FUNCTION_BLOCK TFCalcoliFuoriIngombriColonne
VAR_INPUT
	Traiettoria : POINTER TO TFTraiettoria;
	WorkSpace : POINTER TO TFMachinePalletizer_WorkSpace;
	WorkFootprint : POINTER TO ARRAY [1..MAXFOOTPRINT] OF TFMachinePalletizer_WorkFootprint; //Ingombri
	WorkPickPoint : POINTER TO ARRAY [1..MAXPICKPOINT] OF TFMachinePalletizer_WorkPickPoint;
	//WorkPickPointState : POINTER TO ARRAY [1..MAXPICKPOINT] OF TFMachinePalletizer_WorkPickPointState;
	WorkArea : POINTER TO ARRAY [1..MAXAREA] OF TFMachinePalletizer_WorkArea;
	WorkAreaState : POINTER TO ARRAY [1..MAXAREA] OF TFMachinePalletizer_WorkAreaState;
	Pallet : POINTER TO ARRAY [1..MAXPALLET] OF TFMachinePalletizer_Pallet;
	Layer : POINTER TO ARRAY [1..MAXLAYER] OF TFMachinePalletizer_Layer;
	Forming : POINTER TO ARRAY [1..MAXFORMING] OF TFMachinePalletizer_FormingForSlab;
	PickPlaceParameters	: POINTER TO TFMachinePalletizer_ParametersFromHMI;
	Mission : POINTER TO TFMachinePalletizer_Mission;
	
	WorkAreaManager : POINTER TO TFWorkAreaManager;
	ModuleAX_X : POINTER TO TFModulePalletizer_Ax;
	ModuleAX_Y : POINTER TO TFModulePalletizer_Ax;
	ModuleAX_Z : POINTER TO TFModulePalletizer_Ax;
	ModuleAX_J : POINTER TO TFModulePalletizer_Ax;
	ModuleAX_K : POINTER TO TFModulePalletizer_Ax;
	AbilitaCalcoloIngombroOttimizzato : BOOL := TRUE; //Abilitazione dell'utilizzo degli ingombri ottimizzati... calcoli in base all'angolo di rotazione della pinza
END_VAR
VAR
	f : INT;
	a : INT;
	P : INT;
	wa : int;
	waDXSX : INT;
	AltezzaDiIngombroArea : REAL;
	AltezzaDiIngombroOstacoli : REAL;
	AltezzaDiIngombroPuntiPrelievo : REAL;
	AssegnaQuote : BOOL;
	
	LunghezzaMAX 	: LREAL;//LunghezzaMAX Totale pinza
	LarghezzaMAX 	: LREAL;//Larghezza Totale pinza
	SpessoreMAX  	: LREAL;//Spessore Totale pinza

	IngombroX_Pos : LREAL;//Ingombro della pinza nella Metà POSITIVA della pinza lungo X
	IngombroY_Pos : LREAL;//Ingombro della pinza nella Metà POSITIVA della pinza lungo Y
	
	IngombroX_Neg : LREAL;//Ingombro della pinza nella Metà NEGATIVA della pinza lungo X
	IngombroY_Neg : LREAL;//Ingombro della pinza nella Metà NEGATIVA della pinza lungo Y
	
	IngombroZ : LREAL;//Ingombro della pinza lungo Z
	
	IngombroVerticalePinzaMAX : REAL;
	IngombroVerticaleMaxElementi : REAL;
	//DirezioneXPositiva_Dep : BOOL;
	//DirezioneXNegativa_Dep : BOOL;
	//DirezioneXPositiva_Prel : BOOL;
	//DirezioneXNegativa_Prel : BOOL;
	DirezioneZPositiva : BOOL;
	DirezioneZNegativa : BOOL;
	DirezioneXNegativa : BOOL;
	DirezioneXPositiva : BOOL;
	
	
	WASX : UINT;
	WADX : UINT;
	WAPARTENZA : UINT;
	WADESTINAZIONE : UINT;
	LarghezzaPickPoint : REAL;
	
	
	FuoriIngombroYNecessarioTMP : BOOL;
	QuotaX_ConsensoRotazionePinza_RaggiuntaTMP : BOOL;
	ConsensoTraslazioneY_TraColonneTMP : BOOL;
	AsseXInFinestraDiPrelievoPaccoTMP : BOOL;
	AsseJInFinestraDiPrelievoPaccoTMP : BOOL;
	
	OffsetSicurezza_Y : real := 80;
	
	
	Pinza_InIngombroColonne_Partenza: BOOL; //Indica che la posizione della pinza è in ingombro colonne alla partenza del ciclo/ REAL TIME
	IngombroOttimizzatoY_Destinazione: LREAL;
	IngombroOttimizzatoX_Destinazione: LREAL;
	IngombroOttimizzatoX_InPuntoDiPrelievo: LREAL;
	IngombroOttimizzatoY_InPuntoDiPrelievo: LREAL;
	IngombroOttimizzatoY_InPuntoDiDeposito: LREAL;
	IngombroOttimizzatoX_InPuntoDiDeposito: LREAL;
	//Pinza_InIngombroColonne_Attuale: BOOL;
	//Pinza_InIngombroColonne_Destinazione: BOOL;
	AsseJInFinestraDiPrelievoPallet: BOOL;
	AsseXInFinestraDiPrelievoPallet: BOOL;
	AsseYInFinestraDiPrelievoPallet: BOOL;
	AsseXInFinestraDiRiposo: BOOL;
	AsseYInFinestraDiRiposo: BOOL;
	AsseJInFinestraDiRiposo: BOOL;
	AsseXInFinestraDiDestinazione: BOOL;
	AsseJInFinestraDiDestinazione: BOOL;
	AsseYInFinestraDiDestinazione: BOOL;
	IngombroOttimizzatoX_InTransito: LREAL;
	IngombroOttimizzatoY_InTransito: LREAL;
	Pinza_InIngombroColonne_Transito: BOOL;
	Angolo: INT;
	CalcolaIngombro: BOOL;
	AsseXInFinestraDiPrelievo: BOOL;
	AsseYInFinestraDiPrelievo: BOOL;
	AsseJInFinestraDiPrelievo: BOOL;
	
	QuotaFuoriIngombro_Attuale_Y 		: LREAL;
	QuotaFuoriIngombro_Prelievo_Y 		: LREAL;
	QuotaFuoriIngombro_Deposito_Y		: LREAL;
	
	TFCalcolaQuotaIngombroColonne : TFCalcolaQuotaIngombroColonne;
	TFCalcoloIngombroOttimizzatoPinza : TFCalcoloIngombroOttimizzatoPinza;
	QuotaFuoriIngombro_Destinazione_Y: LREAL;
	WorkAreaManagerState_OLD: INT;
END_VAR

(* Calcolo delle dimensioni della pinza in base al tipo di ciclo in corso *)
CASE WorkAreaManager^.State OF
	WAMANAGER_NOP,
	
	WAMANAGER_CICLO_RIPOSO_INIT,
		
	WAMANAGER_CICLO_RIPOSO_RUN:
		
		SpessoreMAX 	:= Dimensioni_Pinza.Spessore;
		LunghezzaMAX 	:= Dimensioni_Pinza.Lunghezza;
		LarghezzaMAX    := Dimensioni_Pinza.Larghezza;
						
		IngombroX_Pos 	:=  LunghezzaMAX/2;
		IngombroX_Neg 	:=  LunghezzaMAX/2;

		IngombroY_Pos 	:= ABS(LarghezzaMAX/2 * COS(deg_to_rad(90+ModuleAX_J^.Ax^.AxRef^.NcToPlc.ActPos)) +
							SpessoreMAX * SIN(deg_to_rad(90+ModuleAX_J^.Ax^.AxRef^.NcToPlc.ActPos)));
							
		IngombroY_Neg 	:= ABS(LarghezzaMAX/2 * COS(deg_to_rad(90+ModuleAX_J^.Ax^.AxRef^.NcToPlc.ActPos)) -
							SpessoreMAX * SIN(deg_to_rad(90+ModuleAX_J^.Ax^.AxRef^.NcToPlc.ActPos)));	

		IngombroZ		:= Dimensioni_Pinza.Larghezza/2 * SIN(deg_to_rad(90+ModuleAX_J^.Ax^.AxRef^.NcToPlc.ActPos)) +
							SpessoreMAX * COS(deg_to_rad(90+ModuleAX_J^.Ax^.AxRef^.NcToPlc.ActPos));		
									
	WAMANAGER_CICLO_PRELIEVO_FALDA_RUN:
	
		SpessoreMAX 	:= Dimensioni_Pinza.Spessore;
		LunghezzaMAX 	:= Dimensioni_Pinza.Lunghezza;
		LarghezzaMAX    := Dimensioni_Pinza.Larghezza;
						
		IngombroX_Pos 	:=  LunghezzaMAX/2;
		IngombroX_Neg 	:=  LunghezzaMAX/2;

		IngombroY_Pos 	:= ABS(LarghezzaMAX/2 * COS(deg_to_rad(90+ModuleAX_J^.Ax^.AxRef^.NcToPlc.ActPos)) +
							SpessoreMAX * SIN(deg_to_rad(90+ModuleAX_J^.Ax^.AxRef^.NcToPlc.ActPos)));
							
		IngombroY_Neg 	:= ABS(LarghezzaMAX/2 * COS(deg_to_rad(90+ModuleAX_J^.Ax^.AxRef^.NcToPlc.ActPos)) -
							SpessoreMAX * SIN(deg_to_rad(90+ModuleAX_J^.Ax^.AxRef^.NcToPlc.ActPos)));	

		IngombroZ		:= Dimensioni_Pinza.Larghezza/2 * SIN(deg_to_rad(90+ModuleAX_J^.Ax^.AxRef^.NcToPlc.ActPos)) +
							SpessoreMAX * COS(deg_to_rad(90+ModuleAX_J^.Ax^.AxRef^.NcToPlc.ActPos));

	WAMANAGER_CICLO_DEPOSITO_FALDA_RUN:
		
		SpessoreMAX 	:= Dimensioni_Pinza.Spessore;
		LunghezzaMAX 	:= MAX(Dimensioni_Pinza.Lunghezza,Mission^.XDim);
		LarghezzaMAX    := MAX(Dimensioni_Pinza.Larghezza,Mission^.YDim);
						
		IngombroX_Pos 	:=  LunghezzaMAX/2;
		IngombroX_Neg 	:=  LunghezzaMAX/2;

		IngombroY_Pos 	:= ABS(LarghezzaMAX/2 * COS(deg_to_rad(90+ModuleAX_J^.Ax^.AxRef^.NcToPlc.ActPos)) +
							SpessoreMAX * SIN(deg_to_rad(90+ModuleAX_J^.Ax^.AxRef^.NcToPlc.ActPos)));
							
		IngombroY_Neg 	:= ABS(LarghezzaMAX/2 * COS(deg_to_rad(90+ModuleAX_J^.Ax^.AxRef^.NcToPlc.ActPos)) -
							SpessoreMAX * SIN(deg_to_rad(90+ModuleAX_J^.Ax^.AxRef^.NcToPlc.ActPos)));	

		IngombroZ		:= Dimensioni_Pinza.Larghezza/2 * SIN(deg_to_rad(90+ModuleAX_J^.Ax^.AxRef^.NcToPlc.ActPos)) +
							SpessoreMAX * COS(deg_to_rad(90+ModuleAX_J^.Ax^.AxRef^.NcToPlc.ActPos));		
									
				
	WAMANAGER_CICLO_PRELIEVO_LASTRA_WA_RUN:
	
		SpessoreMAX 	:= Dimensioni_Pinza.Spessore;
		LunghezzaMAX 	:= Dimensioni_Pinza.Lunghezza;
		LarghezzaMAX    := Dimensioni_Pinza.Larghezza;
						
		IngombroX_Pos 	:=  LunghezzaMAX/2;
		IngombroX_Neg 	:=  LunghezzaMAX/2;

		IngombroY_Pos 	:= ABS(LarghezzaMAX/2 * COS(deg_to_rad(90+ModuleAX_J^.Ax^.AxRef^.NcToPlc.ActPos)) +
							SpessoreMAX * SIN(deg_to_rad(90+ModuleAX_J^.Ax^.AxRef^.NcToPlc.ActPos)));
							
		IngombroY_Neg 	:= ABS(LarghezzaMAX/2 * COS(deg_to_rad(90+ModuleAX_J^.Ax^.AxRef^.NcToPlc.ActPos)) -
							SpessoreMAX * SIN(deg_to_rad(90+ModuleAX_J^.Ax^.AxRef^.NcToPlc.ActPos)));	

		IngombroZ		:= Dimensioni_Pinza.Larghezza/2 * SIN(deg_to_rad(90+ModuleAX_J^.Ax^.AxRef^.NcToPlc.ActPos)) +
							SpessoreMAX * COS(deg_to_rad(90+ModuleAX_J^.Ax^.AxRef^.NcToPlc.ActPos));
					
	WAMANAGER_CICLO_DEPOSITO_LASTRA_SU_PAREGGIATORE_RUN:
	
		SpessoreMAX 	:= Dimensioni_Pinza.Spessore;
		LunghezzaMAX 	:= MAX(Dimensioni_Pinza.Lunghezza,Mission^.XDim);
		LarghezzaMAX    := MAX(Dimensioni_Pinza.Larghezza,Mission^.YDim);
						
		IngombroX_Pos 	:=  LunghezzaMAX/2;
		IngombroX_Neg 	:=  LunghezzaMAX/2;

		IngombroY_Pos 	:= ABS(LarghezzaMAX/2 * COS(deg_to_rad(90+ModuleAX_J^.Ax^.AxRef^.NcToPlc.ActPos)) +
							SpessoreMAX * SIN(deg_to_rad(90+ModuleAX_J^.Ax^.AxRef^.NcToPlc.ActPos)));
							
		IngombroY_Neg 	:= ABS(LarghezzaMAX/2 * COS(deg_to_rad(90+ModuleAX_J^.Ax^.AxRef^.NcToPlc.ActPos)) -
							SpessoreMAX * SIN(deg_to_rad(90+ModuleAX_J^.Ax^.AxRef^.NcToPlc.ActPos)));	

		IngombroZ		:= Dimensioni_Pinza.Larghezza/2 * SIN(deg_to_rad(90+ModuleAX_J^.Ax^.AxRef^.NcToPlc.ActPos)) +
							SpessoreMAX * COS(deg_to_rad(90+ModuleAX_J^.Ax^.AxRef^.NcToPlc.ActPos));
					
	WAMANAGER_CICLO_PRELIEVO_LASTRA_DA_PAREGGIATORE_RUN:
	
		SpessoreMAX 	:= Dimensioni_Pinza.Spessore;
		LunghezzaMAX 	:= Dimensioni_Pinza.Lunghezza;
		LarghezzaMAX    := Dimensioni_Pinza.Larghezza;
						
		IngombroX_Pos 	:=  LunghezzaMAX/2;
		IngombroX_Neg 	:=  LunghezzaMAX/2;

		IngombroY_Pos 	:= ABS(LarghezzaMAX/2 * COS(deg_to_rad(90+ModuleAX_J^.Ax^.AxRef^.NcToPlc.ActPos)) +
							SpessoreMAX * SIN(deg_to_rad(90+ModuleAX_J^.Ax^.AxRef^.NcToPlc.ActPos)));
							
		IngombroY_Neg 	:= ABS(LarghezzaMAX/2 * COS(deg_to_rad(90+ModuleAX_J^.Ax^.AxRef^.NcToPlc.ActPos)) -
							SpessoreMAX * SIN(deg_to_rad(90+ModuleAX_J^.Ax^.AxRef^.NcToPlc.ActPos)));	

		IngombroZ		:= Dimensioni_Pinza.Larghezza/2 * SIN(deg_to_rad(90+ModuleAX_J^.Ax^.AxRef^.NcToPlc.ActPos)) +
							SpessoreMAX * COS(deg_to_rad(90+ModuleAX_J^.Ax^.AxRef^.NcToPlc.ActPos));				
					
	WAMANAGER_CICLO_DEPOSITO_LASTRA_WA_RUN:
	
		SpessoreMAX 	:= Dimensioni_Pinza.Spessore;
		LunghezzaMAX 	:= MAX(Dimensioni_Pinza.Lunghezza,Mission^.XDim);
		LarghezzaMAX    := MAX(Dimensioni_Pinza.Larghezza,Mission^.YDim);
						
		IngombroX_Pos 	:=  LunghezzaMAX/2;
		IngombroX_Neg 	:=  LunghezzaMAX/2;

		IngombroY_Pos 	:= ABS(LarghezzaMAX/2 * COS(deg_to_rad(90+ModuleAX_J^.Ax^.AxRef^.NcToPlc.ActPos)) +
							SpessoreMAX * SIN(deg_to_rad(90+ModuleAX_J^.Ax^.AxRef^.NcToPlc.ActPos)));
							
		IngombroY_Neg 	:= ABS(LarghezzaMAX/2 * COS(deg_to_rad(90+ModuleAX_J^.Ax^.AxRef^.NcToPlc.ActPos)) -
							SpessoreMAX * SIN(deg_to_rad(90+ModuleAX_J^.Ax^.AxRef^.NcToPlc.ActPos)));	

		IngombroZ		:= Dimensioni_Pinza.Larghezza/2 * SIN(deg_to_rad(90+ModuleAX_J^.Ax^.AxRef^.NcToPlc.ActPos)) +
							SpessoreMAX * COS(deg_to_rad(90+ModuleAX_J^.Ax^.AxRef^.NcToPlc.ActPos));

	WAMANAGER_CICLO_PRELIEVO_LASTRA_PP_RUN:
	
		SpessoreMAX 	:= Dimensioni_Pinza.Spessore;
		LunghezzaMAX 	:= Dimensioni_Pinza.Lunghezza;
		LarghezzaMAX    := Dimensioni_Pinza.Larghezza;
						
		IngombroX_Pos 	:=  LunghezzaMAX/2;
		IngombroX_Neg 	:=  LunghezzaMAX/2;

		IngombroY_Pos 	:= ABS(LarghezzaMAX/2 * COS(deg_to_rad(90+ModuleAX_J^.Ax^.AxRef^.NcToPlc.ActPos)) +
							SpessoreMAX * SIN(deg_to_rad(90+ModuleAX_J^.Ax^.AxRef^.NcToPlc.ActPos)));
							
		IngombroY_Neg 	:= ABS(LarghezzaMAX/2 * COS(deg_to_rad(90+ModuleAX_J^.Ax^.AxRef^.NcToPlc.ActPos)) -
							SpessoreMAX * SIN(deg_to_rad(90+ModuleAX_J^.Ax^.AxRef^.NcToPlc.ActPos)));	

		IngombroZ		:= Dimensioni_Pinza.Larghezza/2 * SIN(deg_to_rad(90+ModuleAX_J^.Ax^.AxRef^.NcToPlc.ActPos)) +
							SpessoreMAX * COS(deg_to_rad(90+ModuleAX_J^.Ax^.AxRef^.NcToPlc.ActPos));			

	WAMANAGER_CICLO_DEPOSITO_LASTRA_PP_RUN:
	
		SpessoreMAX 	:= Dimensioni_Pinza.Spessore;
		LunghezzaMAX 	:= MAX(Dimensioni_Pinza.Lunghezza,Mission^.XDim);
		LarghezzaMAX    := MAX(Dimensioni_Pinza.Larghezza,Mission^.YDim);
						
		IngombroX_Pos 	:=  LunghezzaMAX/2;
		IngombroX_Neg 	:=  LunghezzaMAX/2;

		IngombroY_Pos 	:= ABS(LarghezzaMAX/2 * COS(deg_to_rad(90+ModuleAX_J^.Ax^.AxRef^.NcToPlc.ActPos)) +
							SpessoreMAX * SIN(deg_to_rad(90+ModuleAX_J^.Ax^.AxRef^.NcToPlc.ActPos)));
							
		IngombroY_Neg 	:= ABS(LarghezzaMAX/2 * COS(deg_to_rad(90+ModuleAX_J^.Ax^.AxRef^.NcToPlc.ActPos)) -
							SpessoreMAX * SIN(deg_to_rad(90+ModuleAX_J^.Ax^.AxRef^.NcToPlc.ActPos)));	

		IngombroZ		:= Dimensioni_Pinza.Larghezza/2 * SIN(deg_to_rad(90+ModuleAX_J^.Ax^.AxRef^.NcToPlc.ActPos)) +
							SpessoreMAX * COS(deg_to_rad(90+ModuleAX_J^.Ax^.AxRef^.NcToPlc.ActPos));						
	
END_CASE
(**********************************************************************************************)
(**********************************************************************************************)
(* Setto la variabile per eseguire i calcoli al cambio del WAMANAGER *)
IF WorkAreaManager^.State <> WorkAreaManagerState_OLD THEN
	WorkAreaManagerState_OLD := WorkAreaManager^.State;
	CalcolaIngombro := TRUE; 
END_IF

CASE WorkAreaManager^.State OF
	WAMANAGER_NOP:;
	
	WAMANAGER_CICLO_RIPOSO_INIT:;
		
	WAMANAGER_CICLO_RIPOSO_RUN:
	
		DirezioneXPositiva := TFDirezioneAssePositiva(Posizione_Attuale:=ModuleAX_X^.Ax^.Status.ActPosition,Posizione_Finale:=Mission^.XPick);
		DirezioneXNegativa := NOT DirezioneXPositiva;
		(* Valuto se con l'asse X sono fuori dall'area delle colonne *)
		QuotaX_ConsensoRotazionePinza_Raggiunta := TFPinzaInFuoriIngombroColonne_DirezioneX(DirezioneXPositiva:=DirezioneXPositiva,
																							AsseInMoto:=ModuleAX_X^.Ax^.AxRef^.Status.Moving,
																							PosizioneAttuale:=ModuleAX_X^.Ax^.Status.ActPosition,
																							PosizioneColonna_X:=WorkFootprint^[5].X,  
																							IngombroColonna_X:=WorkFootprint^[5].XDim,
																							IngombroX_Pos:=IngombroX_Pos,
																							IngombroX_Neg:=IngombroX_Neg);
		IF CalcolaIngombro THEN
			CalcolaIngombro := FALSE;
			(* Definisco il tipo di area in cui si trova a lavorare il pallettizzatore *)
			AreaInLavoroPositiva := FALSE;
			AreaInLavoroNegativa := FALSE;
			AreaInLavoroPositivaNegativa := TRUE; 
									
			(**************************************************************************************************************************************************)
			(* Valuto la direzione della X *)
			(**************************************************************************************************************************************************)
			DirezioneXPositiva := TFDirezioneAssePositiva(Posizione_Attuale:=ModuleAX_X^.Ax^.Status.ActPosition,Posizione_Finale:=Mission^.XPick);
			DirezioneXNegativa := NOT DirezioneXPositiva;
			
			(**************************************************************************************************************************************************)
			(* Valuto la direzione della X *)
			(**************************************************************************************************************************************************)
						
			(**************************************************************************************************************************************************)
			(* Ingombro MASSIMO della pinza durante il transito *)
			(**************************************************************************************************************************************************)
			//Calcolo ingombro attuale
			IF NOT TFAsseInFinestra(Posizione_Attuale:=ModuleAx_J^.Ax^.AxRef^.NcToPlc.ActPos,Posizione_Finale:=Mission^.JPick,FinestraDiControllo:=5) THEN //Se la pinza non è già nella finestra di destinazione 
				(* Calcolo l'ingombro massimo che assume durante il ciclo di lavoro nelle direzioni X e Y *)
				(*TFCalcoloIngombroOttimizzatoPinza(  Quota_RotazioneAttuale			:= ModuleAx_J^.Ax^.AxRef^.NcToPlc.ActPos,
													Quota_RotazioneDestinazione		:= Mission^.JPick,
													IngombroSuperficialePinzaMAX	:= IngombroSuperficialePinzaMAX,
													Lunghezza						:= Larghezza,
													Larghezza						:= Lunghezza,
													IngombroOttimizzatoX_InTransito	=> IngombroOttimizzatoX_InTransito,
													IngombroOttimizzatoY_InTransito	=> IngombroOttimizzatoY_InTransito);*)
			ELSE;
				//IngombroOttimizzatoX_InTransito := ABS(IngombroSuperficialePinzaMAX * SIN(deg_to_rad((ATAN(Larghezza/Lunghezza)*1/0.017+ ModuleAx_J^.Ax^.AxRef^.NcToPlc.ActPos)))); //Ingombro Attuale direzione X
				//IngombroOttimizzatoY_InTransito := ABS(IngombroSuperficialePinzaMAX * COS(deg_to_rad((ATAN(Larghezza/Lunghezza)*1/0.017+ ModuleAx_J^.Ax^.AxRef^.NcToPlc.ActPos)))); //Ingombro Attuale direzione Y		
			END_IF
			(* Valutazione colonne in base al verso del pallettizzatore: verso stabilito guardando il pallettizzatore con la linea alle spalle *)
			CASE VERSO_PALLETTIZZATORE OF
				PALLETTIZZATORE_DX :
									TFCalcolaQuotaIngombroColonne(	QuotaY_ColonnaDX						:= WorkFootprint^[6].Y, //DX
																	QuotaY_ColonnaSX						:= WorkFootprint^[5].Y, //SX
																	QuotaAttualeAsse						:= ModuleAX_Y^.Ax^.AxRef^.NcToPlc.ActPos,
																	IngombroOttimizzatoY_InTransito         := IngombroOttimizzatoY_InTransito,
																	OffsetSicurezza_Y						:= OffsetSicurezza_Y,
																	QuotaDestinazioneAsse					:= Mission^.YPick,
																	Pinza_InIngombroColonne_Attuale 		=> Pinza_InIngombroColonne_Attuale,
																	Pinza_InIngombroColonne_Destinazione 	=> Pinza_InIngombroColonne_Destinazione,
																	QuotaFuoriIngombro_Attuale_Y 			=> QuotaFuoriIngombro_Attuale_Y,
																	QuotaFuoriIngombro_Destinazione_Y 		=> QuotaFuoriIngombro_Destinazione_Y);
																	
				PALLETTIZZATORE_SX :
									TFCalcolaQuotaIngombroColonne(	QuotaY_ColonnaDX						:= WorkFootprint^[6].Y, //DX
																	QuotaY_ColonnaSX						:= WorkFootprint^[5].Y, //SX
																	QuotaAttualeAsse						:= ModuleAX_Y^.Ax^.AxRef^.NcToPlc.ActPos,
																	OffsetSicurezza_Y						:= OffsetSicurezza_Y,
																	IngombroOttimizzatoY_InTransito         := IngombroOttimizzatoY_InTransito,
																	QuotaDestinazioneAsse					:= Mission^.YPick,
																	Pinza_InIngombroColonne_Attuale 		=> Pinza_InIngombroColonne_Attuale,
																	Pinza_InIngombroColonne_Destinazione 	=> Pinza_InIngombroColonne_Destinazione,
																	QuotaFuoriIngombro_Attuale_Y 			=> QuotaFuoriIngombro_Attuale_Y,
																	QuotaFuoriIngombro_Destinazione_Y 		=> QuotaFuoriIngombro_Destinazione_Y);
			END_CASE
			
			(* Setto la quota di fuori ingombro che la pinza dovrà assumere durante la traslazione per evitare la collisione con le colonne *)	
			//IF Pinza_InIngombroColonne_Attuale THEN
				QuotaFuoriIngombroColonne_Y := QuotaFuoriIngombro_Attuale_Y;
			//ELSIF Pinza_InIngombroColonne_Destinazione THEN
			//	QuotaFuoriIngombroColonne_Y := QuotaFuoriIngombro_Destinazione_Y;
			//ELSE
			//	QuotaFuoriIngombroColonne_Y := QuotaFuoriIngombro_Attuale_Y;
			//END_IF
			
					
			(* Se sono in ingombro nella posizione attuale o nella posizione di destinazione, devo andare fuori-ingombro con la Y *)
			IF (Pinza_InIngombroColonne_Attuale OR Pinza_InIngombroColonne_Destinazione) THEN 
				IF (AsseXInFinestraDiRiposo AND AsseYInFinestraDiRiposo AND AsseJInFinestraDiRiposo) THEN //Se sono in finestra di riposo con tutti gli assi non devo andare fuori-ingombro con la Y
					FuoriIngombroYNecessarioTMP := FALSE;
				ELSE
					FuoriIngombroYNecessarioTMP := TRUE;
				END_IF
			ELSE
				FuoriIngombroYNecessarioTMP := FALSE;
			END_IF
		END_IF
								
	WAMANAGER_CICLO_RIPOSO_END: 
		CalcolaIngombro := TRUE;
(*			
	WAMANAGER_CICLO_PALL_INIT:
		CalcolaIngombro := TRUE;
	
	WAMANAGER_CICLO_PRELIEVO_PALL_RUN:
		DirezioneXPositiva := TFDirezioneAssePositiva(Posizione_Attuale:=ModuleAX_X^.Ax^.Status.ActPosition,Posizione_Finale:=Mission^.XPick);
		DirezioneXNegativa := NOT DirezioneXPositiva;
		(* Valuto se con l'asse X sono fuori dall'area delle colonne *)
		QuotaX_ConsensoRotazionePinza_Raggiunta := TFPinzaInFuoriIngombroColonne_DirezioneX(DirezioneXPositiva:=DirezioneXPositiva,
																							AsseInMoto:=ModuleAX_X^.Ax^.AxRef^.Status.Moving,
																							PosizioneAttuale:=ModuleAX_X^.Ax^.Status.ActPosition,
																							PosizioneColonna_X:=WorkFootprint^[5].X,  
																							IngombroColonna_X:=WorkFootprint^[5].XDim,
																							IngombroPinza_X:=IngombroX);
				
		IF CalcolaIngombro THEN
			CalcolaIngombro := FALSE;
			(* Definisco il tipo di area in cui si trova a lavorare il pallettizzatore *)
			AreaInLavoroPositiva := FALSE;
			AreaInLavoroNegativa := FALSE;
			AreaInLavoroPositivaNegativa := FALSE; 

			IF (WorkArea^[Mission^.PPick].X >= (WorkFootprint^[5].X + WorkFootprint^[5].XDim)) AND 				//se la piazzola di prelievo è nella campata POSITIVA
				(ModuleAX_X^.Ax^.Status.ActPosition >= (WorkFootprint^[5].X + WorkFootprint^[5].XDim)) THEN // Se la posizione attuale è nella campata POSITIVA
					AreaInLavoroPositiva := TRUE;
			ELSIF (WorkArea^[Mission^.PPick].X <= WorkFootprint^[5].X) AND 			//se la piazzola di prelievo è nella campata NEGATIVA
				(ModuleAX_X^.Ax^.Status.ActPosition <= WorkFootprint^[5].X) THEN 		// Se la posizione attuale è nella campata NEGATIVA
					AreaInLavoroNegativa := TRUE;
			ELSE
				AreaInLavoroPositivaNegativa := TRUE;
			END_IF	
			
			(**************************************************************************************************************************************************)
			(* Ingombro ottimizzato della pinza sul punto di prelievo *)
			(**************************************************************************************************************************************************)
			IngombroOttimizzatoX_InPuntoDiPrelievo := ABS(IngombroSuperficialePinzaMAX * SIN(deg_to_rad((ATAN(Larghezza/Lunghezza)*1/0.017+ Mission^.JPick))));
			IngombroOttimizzatoY_InPuntoDiPrelievo := ABS(IngombroSuperficialePinzaMAX * COS(deg_to_rad((ATAN(Larghezza/Lunghezza)*1/0.017+ Mission^.JPick))));
			(**************************************************************************************************************************************************)
			(* Ingombro ottimizzato della pinza sul punto di deposito *)
			(**************************************************************************************************************************************************)
			IngombroOttimizzatoX_InPuntoDiDeposito := ABS(IngombroSuperficialePinzaMAX * SIN(deg_to_rad((ATAN(Larghezza/Lunghezza)*1/0.017+ Mission^.JPlace))));
			IngombroOttimizzatoY_InPuntoDiDeposito := ABS(IngombroSuperficialePinzaMAX * COS(deg_to_rad((ATAN(Larghezza/Lunghezza)*1/0.017+ Mission^.JPlace))));
						
			(**************************************************************************************************************************************************)
			(**************************************************************************************************************************************************)
			(* Valuto la direzione della X *)
			DirezioneXPositiva := TFDirezioneAssePositiva(Posizione_Attuale:=ModuleAX_X^.Ax^.Status.ActPosition,Posizione_Finale:=Mission^.XPick);
			DirezioneXNegativa := NOT DirezioneXPositiva;
							
			(**************************************************************************************************************************************************)
			(* Ingombro MASSIMO della pinza durante il transito *)
			(**************************************************************************************************************************************************)
			//Calcolo ingombro attuale
			IF NOT TFAsseInFinestra(Posizione_Attuale:=ModuleAx_J^.Ax^.AxRef^.NcToPlc.ActPos,Posizione_Finale:=Mission^.JPick,FinestraDiControllo:=5)  THEN //Se la pinza non è già nella finestra di destinazione 
				(* Calcolo l'ingombro massimo che assume durante il ciclo di lavoro nelle direzioni X e Y *)
				TFCalcoloIngombroOttimizzatoPinza(  Quota_RotazioneAttuale			:= ModuleAx_J^.Ax^.AxRef^.NcToPlc.ActPos,
													Quota_RotazioneDestinazione		:= Mission^.JPick,
													IngombroSuperficialePinzaMAX	:= IngombroSuperficialePinzaMAX,
													Lunghezza						:= Larghezza,
													Larghezza						:= Lunghezza,
													IngombroOttimizzatoX_InTransito	=> IngombroOttimizzatoX_InTransito,
													IngombroOttimizzatoY_InTransito	=> IngombroOttimizzatoY_InTransito);
			ELSE
				IngombroOttimizzatoX_InTransito := ABS(IngombroSuperficialePinzaMAX * SIN(deg_to_rad((ATAN(Larghezza/Lunghezza)*1/0.017+ ModuleAx_J^.Ax^.AxRef^.NcToPlc.ActPos)))); //Ingombro Attuale direzione X
				IngombroOttimizzatoY_InTransito := ABS(IngombroSuperficialePinzaMAX * COS(deg_to_rad((ATAN(Larghezza/Lunghezza)*1/0.017+ ModuleAx_J^.Ax^.AxRef^.NcToPlc.ActPos)))); //Ingombro Attuale direzione Y		
			END_IF
			(* Valutazione colonne in base al verso del pallettizzatore: verso stabilito guardando il pallettizzatore con la linea alle spalle *)
			CASE VERSO_PALLETTIZZATORE OF
				PALLETTIZZATORE_DX :
									TFCalcolaQuotaIngombroColonne(	QuotaY_ColonnaDX						:= WorkFootprint^[6].Y, //DX
																	QuotaY_ColonnaSX						:= WorkFootprint^[5].Y, //SX
																	QuotaAttualeAsse						:= ModuleAX_Y^.Ax^.AxRef^.NcToPlc.ActPos,
																	IngombroOttimizzatoY_InTransito         := IngombroOttimizzatoY_InTransito,
																	OffsetSicurezza_Y						:= OffsetSicurezza_Y,
																	QuotaDestinazioneAsse					:= Mission^.YPick,
																	Pinza_InIngombroColonne_Attuale 		=> Pinza_InIngombroColonne_Attuale,
																	Pinza_InIngombroColonne_Destinazione 	=> Pinza_InIngombroColonne_Destinazione,
																	QuotaFuoriIngombro_Attuale_Y 			=> QuotaFuoriIngombro_Attuale_Y,
																	QuotaFuoriIngombro_Destinazione_Y 		=> QuotaFuoriIngombro_Destinazione_Y);
																	
				PALLETTIZZATORE_SX :
									TFCalcolaQuotaIngombroColonne(	QuotaY_ColonnaDX						:= WorkFootprint^[6].Y, //DX
																	QuotaY_ColonnaSX						:= WorkFootprint^[5].Y, //SX
																	QuotaAttualeAsse						:= ModuleAX_Y^.Ax^.AxRef^.NcToPlc.ActPos,
																	OffsetSicurezza_Y						:= OffsetSicurezza_Y,
																	IngombroOttimizzatoY_InTransito         := IngombroOttimizzatoY_InTransito,
																	QuotaDestinazioneAsse					:= Mission^.YPick,
																	Pinza_InIngombroColonne_Attuale 		=> Pinza_InIngombroColonne_Attuale,
																	Pinza_InIngombroColonne_Destinazione 	=> Pinza_InIngombroColonne_Destinazione,
																	QuotaFuoriIngombro_Attuale_Y 			=> QuotaFuoriIngombro_Attuale_Y,
																	QuotaFuoriIngombro_Destinazione_Y 		=> QuotaFuoriIngombro_Destinazione_Y);
			END_CASE
			
			(* Setto la quota di fuori ingombro che la pinza dovrà assumere durante la traslazione per evitare la collisione con le colonne *)	
			QuotaFuoriIngombroColonne_Y := QuotaFuoriIngombro_Attuale_Y;
					
			(* Se sono in ingombro nella posizione attuale o nella posizione di destinazione, devo andare fuori-ingombro con la Y *)
			IF (Pinza_InIngombroColonne_Attuale OR Pinza_InIngombroColonne_Destinazione) THEN 
				IF (AsseXInFinestraDiRiposo AND AsseYInFinestraDiRiposo AND AsseJInFinestraDiRiposo) THEN //Se sono in finestra di riposo con tutti gli assi non devo andare fuori-ingombro con la Y
					FuoriIngombroYNecessarioTMP := FALSE;
				ELSE
					FuoriIngombroYNecessarioTMP := TRUE;
				END_IF
			ELSE
				FuoriIngombroYNecessarioTMP := FALSE;
			END_IF
		END_IF
		
	WAMANAGER_CICLO_PRELIEVO_PALL_END:
		CalcolaIngombro := TRUE;					
		
	WAMANAGER_CICLO_DEPOSITO_PALL_RUN:
		DirezioneXPositiva := TFDirezioneAssePositiva(Posizione_Attuale:=ModuleAX_X^.Ax^.Status.ActPosition,Posizione_Finale:=Mission^.XPlace);
		DirezioneXNegativa := NOT DirezioneXPositiva;
		(* Valuto se con l'asse X sono fuori dall'area delle colonne *)
		QuotaX_ConsensoRotazionePinza_Raggiunta := TFPinzaInFuoriIngombroColonne_DirezioneX(DirezioneXPositiva:=DirezioneXPositiva,
																							AsseInMoto:=ModuleAX_X^.Ax^.AxRef^.Status.Moving,
																							PosizioneAttuale:=ModuleAX_X^.Ax^.Status.ActPosition,
																							PosizioneColonna_X:=WorkFootprint^[5].X,  
																							IngombroColonna_X:=WorkFootprint^[5].XDim,
																							IngombroPinza_X:=IngombroX);
																					
		IF CalcolaIngombro THEN
			CalcolaIngombro := FALSE;
			(* Definisco il tipo di area in cui si trova a lavorare il pallettizzatore *)
			AreaInLavoroPositiva := FALSE;
			AreaInLavoroNegativa := FALSE;
			AreaInLavoroPositivaNegativa := FALSE; 
			
			IF (WorkArea^[Mission^.PPlace].X >= (WorkFootprint^[5].X + WorkFootprint^[5].XDim)) AND 				//se la piazzola di prelievo è nella campata POSITIVA
				(ModuleAX_X^.Ax^.Status.ActPosition >= (WorkFootprint^[5].X + WorkFootprint^[5].XDim)) THEN // Se la posizione attuale è nella campata POSITIVA
					AreaInLavoroPositiva := TRUE;
			ELSIF (WorkArea^[Mission^.PPlace].X <= WorkFootprint^[5].X) AND 			//se la piazzola di prelievo è nella campata NEGATIVA
				(ModuleAX_X^.Ax^.Status.ActPosition <= WorkFootprint^[5].X) THEN 		// Se la posizione attuale è nella campata NEGATIVA
					AreaInLavoroNegativa := TRUE;
			ELSE
				AreaInLavoroPositivaNegativa := TRUE;
			END_IF
			
			(**************************************************************************************************************************************************)
			(* Ingombro ottimizzato della pinza sul punto di prelievo *)
			(**************************************************************************************************************************************************)
			IngombroOttimizzatoX_InPuntoDiPrelievo := ABS(IngombroSuperficialePinzaMAX * SIN(deg_to_rad((ATAN(Larghezza/Lunghezza)*1/0.017+ Mission^.JPick))));
			IngombroOttimizzatoY_InPuntoDiPrelievo := ABS(IngombroSuperficialePinzaMAX * COS(deg_to_rad((ATAN(Larghezza/Lunghezza)*1/0.017+ Mission^.JPick))));
			(**************************************************************************************************************************************************)
			(* Ingombro ottimizzato della pinza sul punto di deposito *)
			(**************************************************************************************************************************************************)
			IngombroOttimizzatoX_InPuntoDiDeposito := ABS(IngombroSuperficialePinzaMAX * SIN(deg_to_rad((ATAN(Larghezza/Lunghezza)*1/0.017+ Mission^.JPlace))));
			IngombroOttimizzatoY_InPuntoDiDeposito := ABS(IngombroSuperficialePinzaMAX * COS(deg_to_rad((ATAN(Larghezza/Lunghezza)*1/0.017+ Mission^.JPlace))));
						
			(**************************************************************************************************************************************************)
			(**************************************************************************************************************************************************)
			(* Valuto la direzione della X *)
			DirezioneXPositiva := TFDirezioneAssePositiva(Posizione_Attuale:=ModuleAX_X^.Ax^.Status.ActPosition,Posizione_Finale:=Mission^.XPlace);
			DirezioneXNegativa := NOT DirezioneXPositiva;
							
			(**************************************************************************************************************************************************)
			(* Ingombro MASSIMO della pinza durante il transito *)
			(**************************************************************************************************************************************************)
			//Calcolo ingombro attuale
			IF NOT TFAsseInFinestra(Posizione_Attuale:=ModuleAx_J^.Ax^.AxRef^.NcToPlc.ActPos,Posizione_Finale:=Mission^.JPlace,FinestraDiControllo:=5)  THEN //Se la pinza non è già nella finestra di destinazione 
				(* Calcolo l'ingombro massimo che assume durante il ciclo di lavoro nelle direzioni X e Y *)
				TFCalcoloIngombroOttimizzatoPinza(  Quota_RotazioneAttuale			:= ModuleAx_J^.Ax^.AxRef^.NcToPlc.ActPos,
													Quota_RotazioneDestinazione		:= Mission^.JPlace,
													IngombroSuperficialePinzaMAX	:= IngombroSuperficialePinzaMAX,
													Lunghezza						:= Larghezza,
													Larghezza						:= Lunghezza,
													IngombroOttimizzatoX_InTransito	=> IngombroOttimizzatoX_InTransito,
													IngombroOttimizzatoY_InTransito	=> IngombroOttimizzatoY_InTransito);
			ELSE
				IngombroOttimizzatoX_InTransito := ABS(IngombroSuperficialePinzaMAX * SIN(deg_to_rad((ATAN(Larghezza/Lunghezza)*1/0.017+ ModuleAx_J^.Ax^.AxRef^.NcToPlc.ActPos)))); //Ingombro Attuale direzione X
				IngombroOttimizzatoY_InTransito := ABS(IngombroSuperficialePinzaMAX * COS(deg_to_rad((ATAN(Larghezza/Lunghezza)*1/0.017+ ModuleAx_J^.Ax^.AxRef^.NcToPlc.ActPos)))); //Ingombro Attuale direzione Y		
			END_IF
			(* Valutazione colonne in base al verso del pallettizzatore: verso stabilito guardando il pallettizzatore con la linea alle spalle *)
			CASE VERSO_PALLETTIZZATORE OF
				PALLETTIZZATORE_DX :
									TFCalcolaQuotaIngombroColonne(	QuotaY_ColonnaDX						:= WorkFootprint^[6].Y, //DX
																	QuotaY_ColonnaSX						:= WorkFootprint^[5].Y, //SX
																	QuotaAttualeAsse						:= ModuleAX_Y^.Ax^.AxRef^.NcToPlc.ActPos,
																	IngombroOttimizzatoY_InTransito         := IngombroOttimizzatoY_InTransito,
																	OffsetSicurezza_Y						:= OffsetSicurezza_Y,
																	QuotaDestinazioneAsse					:= Mission^.YPlace,
																	Pinza_InIngombroColonne_Attuale 		=> Pinza_InIngombroColonne_Attuale,
																	Pinza_InIngombroColonne_Destinazione 	=> Pinza_InIngombroColonne_Destinazione,
																	QuotaFuoriIngombro_Attuale_Y 			=> QuotaFuoriIngombro_Attuale_Y,
																	QuotaFuoriIngombro_Destinazione_Y 		=> QuotaFuoriIngombro_Destinazione_Y);
																	
				PALLETTIZZATORE_SX :
									TFCalcolaQuotaIngombroColonne(	QuotaY_ColonnaDX						:= WorkFootprint^[6].Y, //DX
																	QuotaY_ColonnaSX						:= WorkFootprint^[5].Y, //SX
																	QuotaAttualeAsse						:= ModuleAX_Y^.Ax^.AxRef^.NcToPlc.ActPos,
																	OffsetSicurezza_Y						:= OffsetSicurezza_Y,
																	IngombroOttimizzatoY_InTransito         := IngombroOttimizzatoY_InTransito,
																	QuotaDestinazioneAsse					:= Mission^.YPlace,
																	Pinza_InIngombroColonne_Attuale 		=> Pinza_InIngombroColonne_Attuale,
																	Pinza_InIngombroColonne_Destinazione 	=> Pinza_InIngombroColonne_Destinazione,
																	QuotaFuoriIngombro_Attuale_Y 			=> QuotaFuoriIngombro_Attuale_Y,
																	QuotaFuoriIngombro_Destinazione_Y 		=> QuotaFuoriIngombro_Destinazione_Y);
			END_CASE
			
			(* Setto la quota di fuori ingombro che la pinza dovrà assumere durante la traslazione per evitare la collisione con le colonne *)	
			QuotaFuoriIngombroColonne_Y := QuotaFuoriIngombro_Attuale_Y;
					
			(* Se sono in ingombro nella posizione attuale o nella posizione di destinazione, devo andare fuori-ingombro con la Y *)
			IF (Pinza_InIngombroColonne_Attuale OR Pinza_InIngombroColonne_Destinazione) THEN 
				IF (AsseXInFinestraDiRiposo AND AsseYInFinestraDiRiposo AND AsseJInFinestraDiRiposo) THEN //Se sono in finestra di riposo con tutti gli assi non devo andare fuori-ingombro con la Y
					FuoriIngombroYNecessarioTMP := FALSE;
				ELSE
					FuoriIngombroYNecessarioTMP := TRUE;
				END_IF
			ELSE
				FuoriIngombroYNecessarioTMP := FALSE;
			END_IF
		END_IF
		
	WAMANAGER_CICLO_DEPOSITO_PALL_END:
		CalcolaIngombro := TRUE;	
	
	WAMANAGER_CICLO_FALDA_VUOTI_INIT:
		CalcolaIngombro := TRUE;	
	
	WAMANAGER_CICLO_PRELIEVO_FALDA_VUOTI_RUN:
		DirezioneXPositiva := TFDirezioneAssePositiva(Posizione_Attuale:=ModuleAX_X^.Ax^.Status.ActPosition,Posizione_Finale:=Mission^.XPick);
		DirezioneXNegativa := NOT DirezioneXPositiva;
		
				
		IF CalcolaIngombro THEN
			CalcolaIngombro := FALSE;
			(* Definisco il tipo di area in cui si trova a lavorare il pallettizzatore *)
			AreaInLavoroPositiva := FALSE;
			AreaInLavoroNegativa := FALSE;
			AreaInLavoroPositivaNegativa := FALSE;

			IF (WorkArea^[Mission^.PPick].X >= (WorkFootprint^[5].X + WorkFootprint^[5].XDim)) AND 				//se la piazzola di prelievo è nella campata POSITIVA
				(ModuleAX_X^.Ax^.Status.ActPosition >= (WorkFootprint^[5].X + WorkFootprint^[5].XDim)) THEN // Se la posizione attuale è nella campata POSITIVA
					AreaInLavoroPositiva := TRUE;
			ELSIF (WorkArea^[Mission^.PPick].X <= WorkFootprint^[5].X) AND 			//se la piazzola di prelievo è nella campata NEGATIVA
				(ModuleAX_X^.Ax^.Status.ActPosition <= WorkFootprint^[5].X) THEN 		// Se la posizione attuale è nella campata NEGATIVA
					AreaInLavoroNegativa := TRUE;
			ELSE
				AreaInLavoroPositivaNegativa := TRUE;
			END_IF 
			
			(**************************************************************************************************************************************************)
			(* Ingombro ottimizzato della pinza sul punto di prelievo *)
			(**************************************************************************************************************************************************)
			IngombroOttimizzatoX_InPuntoDiPrelievo := ABS(IngombroSuperficialePinzaMAX * SIN(deg_to_rad((ATAN(Larghezza/Lunghezza)*1/0.017+ Mission^.JPick))));
			IngombroOttimizzatoY_InPuntoDiPrelievo := ABS(IngombroSuperficialePinzaMAX * COS(deg_to_rad((ATAN(Larghezza/Lunghezza)*1/0.017+ Mission^.JPick))));
			(**************************************************************************************************************************************************)
			(* Ingombro ottimizzato della pinza sul punto di deposito *)
			(**************************************************************************************************************************************************)
			IngombroOttimizzatoX_InPuntoDiDeposito := ABS(IngombroSuperficialePinzaMAX * SIN(deg_to_rad((ATAN(Larghezza/Lunghezza)*1/0.017+ Mission^.JPlace))));
			IngombroOttimizzatoY_InPuntoDiDeposito := ABS(IngombroSuperficialePinzaMAX * COS(deg_to_rad((ATAN(Larghezza/Lunghezza)*1/0.017+ Mission^.JPlace))));
						
			(**************************************************************************************************************************************************)
			(**************************************************************************************************************************************************)
			(* Valuto la direzione della X *)
			DirezioneXPositiva := TFDirezioneAssePositiva(Posizione_Attuale:=ModuleAX_X^.Ax^.Status.ActPosition,Posizione_Finale:=Mission^.XPick);
			DirezioneXNegativa := NOT DirezioneXPositiva;
							
			(**************************************************************************************************************************************************)
			(* Ingombro MASSIMO della pinza durante il transito *)
			(**************************************************************************************************************************************************)
			//Calcolo ingombro attuale
			IF NOT TFAsseInFinestra(Posizione_Attuale:=ModuleAx_J^.Ax^.AxRef^.NcToPlc.ActPos,Posizione_Finale:=Mission^.JPick,FinestraDiControllo:=5)  THEN //Se la pinza non è già nella finestra di destinazione 
				(* Calcolo l'ingombro massimo che assume durante il ciclo di lavoro nelle direzioni X e Y *)
				TFCalcoloIngombroOttimizzatoPinza(  Quota_RotazioneAttuale			:= ModuleAx_J^.Ax^.AxRef^.NcToPlc.ActPos,
													Quota_RotazioneDestinazione		:= Mission^.JPick,
													IngombroSuperficialePinzaMAX	:= IngombroSuperficialePinzaMAX,
													Lunghezza						:= Larghezza,
													Larghezza						:= Lunghezza,
													IngombroOttimizzatoX_InTransito	=> IngombroOttimizzatoX_InTransito,
													IngombroOttimizzatoY_InTransito	=> IngombroOttimizzatoY_InTransito);
			ELSE
				IngombroOttimizzatoX_InTransito := ABS(IngombroSuperficialePinzaMAX * SIN(deg_to_rad((ATAN(Larghezza/Lunghezza)*1/0.017+ ModuleAx_J^.Ax^.AxRef^.NcToPlc.ActPos)))); //Ingombro Attuale direzione X
				IngombroOttimizzatoY_InTransito := ABS(IngombroSuperficialePinzaMAX * COS(deg_to_rad((ATAN(Larghezza/Lunghezza)*1/0.017+ ModuleAx_J^.Ax^.AxRef^.NcToPlc.ActPos)))); //Ingombro Attuale direzione Y		
			END_IF
			(* Valutazione colonne in base al verso del pallettizzatore: verso stabilito guardando il pallettizzatore con la linea alle spalle *)
			CASE VERSO_PALLETTIZZATORE OF
				PALLETTIZZATORE_DX :
									TFCalcolaQuotaIngombroColonne(	QuotaY_ColonnaDX						:= WorkFootprint^[6].Y, //DX
																	QuotaY_ColonnaSX						:= WorkFootprint^[5].Y, //SX
																	QuotaAttualeAsse						:= ModuleAX_Y^.Ax^.AxRef^.NcToPlc.ActPos,
																	IngombroOttimizzatoY_InTransito         := IngombroOttimizzatoY_InTransito,
																	OffsetSicurezza_Y						:= OffsetSicurezza_Y,
																	QuotaDestinazioneAsse					:= Mission^.YPick,
																	Pinza_InIngombroColonne_Attuale 		=> Pinza_InIngombroColonne_Attuale,
																	Pinza_InIngombroColonne_Destinazione 	=> Pinza_InIngombroColonne_Destinazione,
																	QuotaFuoriIngombro_Attuale_Y 			=> QuotaFuoriIngombro_Attuale_Y,
																	QuotaFuoriIngombro_Destinazione_Y 		=> QuotaFuoriIngombro_Destinazione_Y);
																	
				PALLETTIZZATORE_SX :
									TFCalcolaQuotaIngombroColonne(	QuotaY_ColonnaDX						:= WorkFootprint^[6].Y, //DX
																	QuotaY_ColonnaSX						:= WorkFootprint^[5].Y, //SX
																	QuotaAttualeAsse						:= ModuleAX_Y^.Ax^.AxRef^.NcToPlc.ActPos,
																	OffsetSicurezza_Y						:= OffsetSicurezza_Y,
																	IngombroOttimizzatoY_InTransito         := IngombroOttimizzatoY_InTransito,
																	QuotaDestinazioneAsse					:= Mission^.YPick,
																	Pinza_InIngombroColonne_Attuale 		=> Pinza_InIngombroColonne_Attuale,
																	Pinza_InIngombroColonne_Destinazione 	=> Pinza_InIngombroColonne_Destinazione,
																	QuotaFuoriIngombro_Attuale_Y 			=> QuotaFuoriIngombro_Attuale_Y,
																	QuotaFuoriIngombro_Destinazione_Y 		=> QuotaFuoriIngombro_Destinazione_Y);
			END_CASE
			
			(* Setto la quota di fuori ingombro che la pinza dovrà assumere durante la traslazione per evitare la collisione con le colonne *)	
			QuotaFuoriIngombroColonne_Y := QuotaFuoriIngombro_Attuale_Y;
					
			(* Se sono in ingombro nella posizione attuale o nella posizione di destinazione, devo andare fuori-ingombro con la Y *)
			IF (Pinza_InIngombroColonne_Attuale OR Pinza_InIngombroColonne_Destinazione) THEN 
				IF (AsseXInFinestraDiRiposo AND AsseYInFinestraDiRiposo AND AsseJInFinestraDiRiposo) THEN //Se sono in finestra di riposo con tutti gli assi non devo andare fuori-ingombro con la Y
					FuoriIngombroYNecessarioTMP := FALSE;
				ELSE
					FuoriIngombroYNecessarioTMP := TRUE;
				END_IF
			ELSE
				FuoriIngombroYNecessarioTMP := FALSE;
			END_IF
		END_IF
		
		(* Valuto se con l'asse X sono fuori dall'area delle colonne *)
		QuotaX_ConsensoRotazionePinza_Raggiunta := NOT AreaInLavoroPositivaNegativa OR TFPinzaInFuoriIngombroColonne_DirezioneX(DirezioneXPositiva:=DirezioneXPositiva,
																							AsseInMoto:=ModuleAX_X^.Ax^.AxRef^.Status.Moving,
																							PosizioneAttuale:=ModuleAX_X^.Ax^.Status.ActPosition,
																							PosizioneColonna_X:=WorkFootprint^[5].X,  
																							IngombroColonna_X:=WorkFootprint^[5].XDim,
																							IngombroPinza_X:=IngombroX);
			
	WAMANAGER_CICLO_PRELIEVO_FALDA_VUOTI_END:
		CalcolaIngombro := TRUE;	
		
	WAMANAGER_CICLO_DEPOSITO_FALDA_VUOTI_RUN:
		DirezioneXPositiva := TFDirezioneAssePositiva(Posizione_Attuale:=ModuleAX_X^.Ax^.Status.ActPosition,Posizione_Finale:=Mission^.XPlace);
		DirezioneXNegativa := NOT DirezioneXPositiva;
		(* Valuto se con l'asse X sono fuori dall'area delle colonne *)
		QuotaX_ConsensoRotazionePinza_Raggiunta := TFPinzaInFuoriIngombroColonne_DirezioneX(DirezioneXPositiva:=DirezioneXPositiva,
																							AsseInMoto:=ModuleAX_X^.Ax^.AxRef^.Status.Moving,
																							PosizioneAttuale:=ModuleAX_X^.Ax^.Status.ActPosition,
																							PosizioneColonna_X:=WorkFootprint^[5].X,  
																							IngombroColonna_X:=WorkFootprint^[5].XDim,
																							IngombroPinza_X:=IngombroX);
				IF CalcolaIngombro THEN
			CalcolaIngombro := FALSE;
			(* Definisco il tipo di area in cui si trova a lavorare il pallettizzatore *)
			AreaInLavoroPositiva := FALSE;
			AreaInLavoroNegativa := FALSE;
			AreaInLavoroPositivaNegativa := FALSE; 
			
			IF (WorkArea^[Mission^.PPlace].X >= (WorkFootprint^[5].X + WorkFootprint^[5].XDim)) AND 		//se la piazzola di prelievo è nella campata POSITIVA
				(ModuleAX_X^.Ax^.Status.ActPosition >= (WorkFootprint^[5].X + WorkFootprint^[5].XDim)) THEN // Se la posizione attuale è nella campata POSITIVA
					AreaInLavoroPositivaNegativa := FALSE; 
					AreaInLavoroPositiva := TRUE;
			ELSIF (WorkArea^[Mission^.PPlace].X <= WorkFootprint^[5].X) AND 			//se la piazzola di prelievo è nella campata NEGATIVA
				(ModuleAX_X^.Ax^.Status.ActPosition <= WorkFootprint^[5].X) THEN 		// Se la posizione attuale è nella campata NEGATIVA
					AreaInLavoroPositivaNegativa := FALSE; 
					AreaInLavoroNegativa := TRUE;
			ELSE
				AreaInLavoroPositivaNegativa := TRUE;
			END_IF
			
			(**************************************************************************************************************************************************)
			(* Ingombro ottimizzato della pinza sul punto di prelievo *)
			(**************************************************************************************************************************************************)
			IngombroOttimizzatoX_InPuntoDiPrelievo := ABS(IngombroSuperficialePinzaMAX * SIN(deg_to_rad((ATAN(Larghezza/Lunghezza)*1/0.017+ Mission^.JPick))));
			IngombroOttimizzatoY_InPuntoDiPrelievo := ABS(IngombroSuperficialePinzaMAX * COS(deg_to_rad((ATAN(Larghezza/Lunghezza)*1/0.017+ Mission^.JPick))));
			(**************************************************************************************************************************************************)
			(* Ingombro ottimizzato della pinza sul punto di deposito *)
			(**************************************************************************************************************************************************)
			IngombroOttimizzatoX_InPuntoDiDeposito := ABS(IngombroSuperficialePinzaMAX * SIN(deg_to_rad((ATAN(Larghezza/Lunghezza)*1/0.017+ Mission^.JPlace))));
			IngombroOttimizzatoY_InPuntoDiDeposito := ABS(IngombroSuperficialePinzaMAX * COS(deg_to_rad((ATAN(Larghezza/Lunghezza)*1/0.017+ Mission^.JPlace))));
						
			(**************************************************************************************************************************************************)
			(**************************************************************************************************************************************************)
			(* Valuto la direzione della X *)
			DirezioneXPositiva := TFDirezioneAssePositiva(Posizione_Attuale:=ModuleAX_X^.Ax^.Status.ActPosition,Posizione_Finale:=Mission^.XPlace);
			DirezioneXNegativa := NOT DirezioneXPositiva;
							
			(**************************************************************************************************************************************************)
			(* Ingombro MASSIMO della pinza durante il transito *)
			(**************************************************************************************************************************************************)
			//Calcolo ingombro attuale
			IF NOT TFAsseInFinestra(Posizione_Attuale:=ModuleAx_J^.Ax^.AxRef^.NcToPlc.ActPos,Posizione_Finale:=Mission^.JPlace,FinestraDiControllo:=5)  THEN //Se la pinza non è già nella finestra di destinazione 
				(* Calcolo l'ingombro massimo che assume durante il ciclo di lavoro nelle direzioni X e Y *)
				TFCalcoloIngombroOttimizzatoPinza(  Quota_RotazioneAttuale			:= ModuleAx_J^.Ax^.AxRef^.NcToPlc.ActPos,
													Quota_RotazioneDestinazione		:= Mission^.JPlace,
													IngombroSuperficialePinzaMAX	:= IngombroSuperficialePinzaMAX,
													Lunghezza						:= Larghezza,
													Larghezza						:= Lunghezza,
													IngombroOttimizzatoX_InTransito	=> IngombroOttimizzatoX_InTransito,
													IngombroOttimizzatoY_InTransito	=> IngombroOttimizzatoY_InTransito);
			ELSE
				IngombroOttimizzatoX_InTransito := ABS(IngombroSuperficialePinzaMAX * SIN(deg_to_rad((ATAN(Larghezza/Lunghezza)*1/0.017+ ModuleAx_J^.Ax^.AxRef^.NcToPlc.ActPos)))); //Ingombro Attuale direzione X
				IngombroOttimizzatoY_InTransito := ABS(IngombroSuperficialePinzaMAX * COS(deg_to_rad((ATAN(Larghezza/Lunghezza)*1/0.017+ ModuleAx_J^.Ax^.AxRef^.NcToPlc.ActPos)))); //Ingombro Attuale direzione Y		
			END_IF
			(* Valutazione colonne in base al verso del pallettizzatore: verso stabilito guardando il pallettizzatore con la linea alle spalle *)
			CASE VERSO_PALLETTIZZATORE OF
				PALLETTIZZATORE_DX :
									TFCalcolaQuotaIngombroColonne(	QuotaY_ColonnaDX						:= WorkFootprint^[6].Y, //DX
																	QuotaY_ColonnaSX						:= WorkFootprint^[5].Y, //SX
																	QuotaAttualeAsse						:= ModuleAX_Y^.Ax^.AxRef^.NcToPlc.ActPos,
																	IngombroOttimizzatoY_InTransito         := IngombroOttimizzatoY_InTransito,
																	OffsetSicurezza_Y						:= OffsetSicurezza_Y,
																	QuotaDestinazioneAsse					:= Mission^.YPlace,
																	Pinza_InIngombroColonne_Attuale 		=> Pinza_InIngombroColonne_Attuale,
																	Pinza_InIngombroColonne_Destinazione 	=> Pinza_InIngombroColonne_Destinazione,
																	QuotaFuoriIngombro_Attuale_Y 			=> QuotaFuoriIngombro_Attuale_Y,
																	QuotaFuoriIngombro_Destinazione_Y 		=> QuotaFuoriIngombro_Destinazione_Y);
																	
				PALLETTIZZATORE_SX :
									TFCalcolaQuotaIngombroColonne(	QuotaY_ColonnaDX						:= WorkFootprint^[6].Y, //DX
																	QuotaY_ColonnaSX						:= WorkFootprint^[5].Y, //SX
																	QuotaAttualeAsse						:= ModuleAX_Y^.Ax^.AxRef^.NcToPlc.ActPos,
																	OffsetSicurezza_Y						:= OffsetSicurezza_Y,
																	IngombroOttimizzatoY_InTransito         := IngombroOttimizzatoY_InTransito,
																	QuotaDestinazioneAsse					:= Mission^.YPlace,
																	Pinza_InIngombroColonne_Attuale 		=> Pinza_InIngombroColonne_Attuale,
																	Pinza_InIngombroColonne_Destinazione 	=> Pinza_InIngombroColonne_Destinazione,
																	QuotaFuoriIngombro_Attuale_Y 			=> QuotaFuoriIngombro_Attuale_Y,
																	QuotaFuoriIngombro_Destinazione_Y 		=> QuotaFuoriIngombro_Destinazione_Y);
			END_CASE
			
			(* Setto la quota di fuori ingombro che la pinza dovrà assumere durante la traslazione per evitare la collisione con le colonne *)	
			QuotaFuoriIngombroColonne_Y := MAX(QuotaFuoriIngombro_Attuale_Y,QuotaFuoriIngombro_Destinazione_Y);
					
			(* Se sono in ingombro nella posizione attuale o nella posizione di destinazione, devo andare fuori-ingombro con la Y *)
			IF (Pinza_InIngombroColonne_Attuale OR Pinza_InIngombroColonne_Destinazione) THEN 
				IF (AsseXInFinestraDiRiposo AND AsseYInFinestraDiRiposo AND AsseJInFinestraDiRiposo) THEN //Se sono in finestra di riposo con tutti gli assi non devo andare fuori-ingombro con la Y
					FuoriIngombroYNecessarioTMP := FALSE;
				ELSE
					FuoriIngombroYNecessarioTMP := TRUE;
				END_IF
			ELSE
				FuoriIngombroYNecessarioTMP := FALSE;
			END_IF
		END_IF
								
	//WAMANAGER_CICLO_DEPOSITO_FALDA_VUOTI_END:
	//	CalcolaIngombro := TRUE;	
	*)
	WAMANAGER_CICLO_FALDA_INIT:
		CalcolaIngombro := TRUE;	
	
	WAMANAGER_CICLO_PRELIEVO_FALDA_RUN:
		DirezioneXPositiva := TFDirezioneAssePositiva(Posizione_Attuale:=ModuleAX_X^.Ax^.Status.ActPosition,Posizione_Finale:=Mission^.XPick);
		DirezioneXNegativa := NOT DirezioneXPositiva;
		(* Valuto se con l'asse X sono fuori dall'area delle colonne *)
		(*QuotaX_ConsensoRotazionePinza_Raggiunta := TFPinzaInFuoriIngombroColonne_DirezioneX(DirezioneXPositiva:=DirezioneXPositiva,
																							AsseInMoto:=ModuleAX_X^.Ax^.AxRef^.Status.Moving,
																							PosizioneAttuale:=ModuleAX_X^.Ax^.Status.ActPosition,
																							PosizioneColonna_X:=WorkFootprint^[5].X,  
																							IngombroColonna_X:=WorkFootprint^[5].XDim,
																							IngombroPinza_X:=IngombroX);*)
																							
		IF CalcolaIngombro THEN
			CalcolaIngombro := FALSE;
			(* Definisco il tipo di area in cui si trova a lavorare il pallettizzatore *)
			AreaInLavoroPositiva := FALSE;
			AreaInLavoroNegativa := FALSE;
			AreaInLavoroPositivaNegativa := FALSE; 
			
			IF (WorkArea^[Mission^.PPick].X >= (WorkFootprint^[5].X + WorkFootprint^[5].XDim)) AND 				//se la piazzola di prelievo è nella campata POSITIVA
				(ModuleAX_X^.Ax^.Status.ActPosition >= (WorkFootprint^[5].X + WorkFootprint^[5].XDim)) THEN // Se la posizione attuale è nella campata POSITIVA
					AreaInLavoroPositiva := TRUE;
			ELSIF (WorkArea^[Mission^.PPick].X <= WorkFootprint^[5].X) AND 			//se la piazzola di prelievo è nella campata NEGATIVA
				(ModuleAX_X^.Ax^.Status.ActPosition <= WorkFootprint^[5].X) THEN 		// Se la posizione attuale è nella campata NEGATIVA
					AreaInLavoroNegativa := TRUE;
			ELSE
				AreaInLavoroPositivaNegativa := TRUE;
			END_IF
			(**************************************************************************************************************************************************)
			(* Ingombro ottimizzato della pinza sul punto di prelievo *)
			(**************************************************************************************************************************************************)
			(*IngombroOttimizzatoX_InPuntoDiPrelievo := ABS(IngombroSuperficialePinzaMAX * SIN(deg_to_rad((ATAN(Larghezza/Lunghezza)*1/0.017+ Mission^.JPick))));
			IngombroOttimizzatoY_InPuntoDiPrelievo := ABS(IngombroSuperficialePinzaMAX * COS(deg_to_rad((ATAN(Larghezza/Lunghezza)*1/0.017+ Mission^.JPick))));
			(**************************************************************************************************************************************************)
			(* Ingombro ottimizzato della pinza sul punto di deposito *)
			(**************************************************************************************************************************************************)
			IngombroOttimizzatoX_InPuntoDiDeposito := ABS(IngombroSuperficialePinzaMAX * SIN(deg_to_rad((ATAN(Larghezza/Lunghezza)*1/0.017+ Mission^.JPlace))));
			IngombroOttimizzatoY_InPuntoDiDeposito := ABS(IngombroSuperficialePinzaMAX * COS(deg_to_rad((ATAN(Larghezza/Lunghezza)*1/0.017+ Mission^.JPlace))));
			*)			
			(**************************************************************************************************************************************************)
			(**************************************************************************************************************************************************)
			(* Valuto la direzione della X *)
			DirezioneXPositiva := TFDirezioneAssePositiva(Posizione_Attuale:=ModuleAX_X^.Ax^.Status.ActPosition,Posizione_Finale:=Mission^.XPick);
			DirezioneXNegativa := NOT DirezioneXPositiva;
							
			(**************************************************************************************************************************************************)
			(* Ingombro MASSIMO della pinza durante il transito *)
			(**************************************************************************************************************************************************)
			//Calcolo ingombro attuale
			IF NOT TFAsseInFinestra(Posizione_Attuale:=ModuleAx_J^.Ax^.AxRef^.NcToPlc.ActPos,Posizione_Finale:=Mission^.JPick,FinestraDiControllo:=5)  THEN //Se la pinza non è già nella finestra di destinazione 
				(* Calcolo l'ingombro massimo che assume durante il ciclo di lavoro nelle direzioni X e Y *)
				(*TFCalcoloIngombroOttimizzatoPinza(  Quota_RotazioneAttuale			:= ModuleAx_J^.Ax^.AxRef^.NcToPlc.ActPos,
													Quota_RotazioneDestinazione		:= Mission^.JPick,
													IngombroSuperficialePinzaMAX	:= IngombroSuperficialePinzaMAX,
													Lunghezza						:= Larghezza,
													Larghezza						:= Lunghezza,
													IngombroOttimizzatoX_InTransito	=> IngombroOttimizzatoX_InTransito,
													IngombroOttimizzatoY_InTransito	=> IngombroOttimizzatoY_InTransito);*)
			ELSE;
				//IngombroOttimizzatoX_InTransito := ABS(IngombroSuperficialePinzaMAX * SIN(deg_to_rad((ATAN(Larghezza/Lunghezza)*1/0.017+ ModuleAx_J^.Ax^.AxRef^.NcToPlc.ActPos)))); //Ingombro Attuale direzione X
				//IngombroOttimizzatoY_InTransito := ABS(IngombroSuperficialePinzaMAX * COS(deg_to_rad((ATAN(Larghezza/Lunghezza)*1/0.017+ ModuleAx_J^.Ax^.AxRef^.NcToPlc.ActPos)))); //Ingombro Attuale direzione Y		
			END_IF
			(* Valutazione colonne in base al verso del pallettizzatore: verso stabilito guardando il pallettizzatore con la linea alle spalle *)
			CASE VERSO_PALLETTIZZATORE OF
				PALLETTIZZATORE_DX :
									TFCalcolaQuotaIngombroColonne(	QuotaY_ColonnaDX						:= WorkFootprint^[6].Y, //DX
																	QuotaY_ColonnaSX						:= WorkFootprint^[5].Y, //SX
																	QuotaAttualeAsse						:= ModuleAX_Y^.Ax^.AxRef^.NcToPlc.ActPos,
																	IngombroOttimizzatoY_InTransito         := IngombroOttimizzatoY_InTransito,
																	OffsetSicurezza_Y						:= OffsetSicurezza_Y,
																	QuotaDestinazioneAsse					:= Mission^.YPick,
																	Pinza_InIngombroColonne_Attuale 		=> Pinza_InIngombroColonne_Attuale,
																	Pinza_InIngombroColonne_Destinazione 	=> Pinza_InIngombroColonne_Destinazione,
																	QuotaFuoriIngombro_Attuale_Y 			=> QuotaFuoriIngombro_Attuale_Y,
																	QuotaFuoriIngombro_Destinazione_Y 		=> QuotaFuoriIngombro_Destinazione_Y);
																	
				PALLETTIZZATORE_SX :
									TFCalcolaQuotaIngombroColonne(	QuotaY_ColonnaDX						:= WorkFootprint^[6].Y, //DX
																	QuotaY_ColonnaSX						:= WorkFootprint^[5].Y, //SX
																	QuotaAttualeAsse						:= ModuleAX_Y^.Ax^.AxRef^.NcToPlc.ActPos,
																	OffsetSicurezza_Y						:= OffsetSicurezza_Y,
																	IngombroOttimizzatoY_InTransito         := IngombroOttimizzatoY_InTransito,
																	QuotaDestinazioneAsse					:= Mission^.YPick,
																	Pinza_InIngombroColonne_Attuale 		=> Pinza_InIngombroColonne_Attuale,
																	Pinza_InIngombroColonne_Destinazione 	=> Pinza_InIngombroColonne_Destinazione,
																	QuotaFuoriIngombro_Attuale_Y 			=> QuotaFuoriIngombro_Attuale_Y,
																	QuotaFuoriIngombro_Destinazione_Y 		=> QuotaFuoriIngombro_Destinazione_Y);
			END_CASE
			
			(* Setto la quota di fuori ingombro che la pinza dovrà assumere durante la traslazione per evitare la collisione con le colonne *)	
			QuotaFuoriIngombroColonne_Y := QuotaFuoriIngombro_Attuale_Y;
					
			(* Se sono in ingombro nella posizione attuale o nella posizione di destinazione, devo andare fuori-ingombro con la Y *)
			IF (Pinza_InIngombroColonne_Attuale OR Pinza_InIngombroColonne_Destinazione) THEN 
				IF (AsseXInFinestraDiRiposo AND AsseYInFinestraDiRiposo AND AsseJInFinestraDiRiposo) THEN //Se sono in finestra di riposo con tutti gli assi non devo andare fuori-ingombro con la Y
					FuoriIngombroYNecessarioTMP := FALSE;
				ELSE
					FuoriIngombroYNecessarioTMP := TRUE;
				END_IF
			ELSE
				FuoriIngombroYNecessarioTMP := FALSE;
			END_IF
		END_IF	
																
	WAMANAGER_CICLO_PRELIEVO_FALDA_END:
		CalcolaIngombro := TRUE;	
			
	WAMANAGER_CICLO_DEPOSITO_FALDA_RUN:
		DirezioneXPositiva := TFDirezioneAssePositiva(Posizione_Attuale:=ModuleAX_X^.Ax^.Status.ActPosition,Posizione_Finale:=Mission^.XPlace);
		DirezioneXNegativa := NOT DirezioneXPositiva;
		(* Valuto se con l'asse X sono fuori dall'area delle colonne *)
		(*QuotaX_ConsensoRotazionePinza_Raggiunta := TFPinzaInFuoriIngombroColonne_DirezioneX(DirezioneXPositiva:=DirezioneXPositiva,
																							AsseInMoto:=ModuleAX_X^.Ax^.AxRef^.Status.Moving,
																							PosizioneAttuale:=ModuleAX_X^.Ax^.Status.ActPosition,
																							PosizioneColonna_X:=WorkFootprint^[5].X,  
																							IngombroColonna_X:=WorkFootprint^[5].XDim,
																							IngombroPinza_X:=IngombroX);*)
																							
		IF (WorkArea^[Mission^.PPlace].X >= (WorkFootprint^[5].X + WorkFootprint^[5].XDim)) AND 				//se la piazzola di prelievo è nella campata POSITIVA
			(ModuleAX_X^.Ax^.Status.ActPosition >= (WorkFootprint^[5].X + WorkFootprint^[5].XDim)) THEN // Se la posizione attuale è nella campata POSITIVA
				AreaInLavoroPositiva := TRUE;
		ELSIF (WorkArea^[Mission^.PPlace].X <= WorkFootprint^[5].X) AND 			//se la piazzola di prelievo è nella campata NEGATIVA
			(ModuleAX_X^.Ax^.Status.ActPosition <= WorkFootprint^[5].X) THEN 		// Se la posizione attuale è nella campata NEGATIVA
				AreaInLavoroNegativa := TRUE;
		ELSE
			AreaInLavoroPositivaNegativa := TRUE;
		END_IF
		
		IF CalcolaIngombro THEN
			CalcolaIngombro := FALSE;
			(* Definisco il tipo di area in cui si trova a lavorare il pallettizzatore *)
			AreaInLavoroPositiva := FALSE;
			AreaInLavoroNegativa := FALSE;
			AreaInLavoroPositivaNegativa := TRUE; 
			
			(**************************************************************************************************************************************************)
			(* Ingombro ottimizzato della pinza sul punto di prelievo *)
			(**************************************************************************************************************************************************)
		(*	IngombroOttimizzatoX_InPuntoDiPrelievo := ABS(IngombroSuperficialePinzaMAX * SIN(deg_to_rad((ATAN(Larghezza/Lunghezza)*1/0.017+ Mission^.JPick))));
			IngombroOttimizzatoY_InPuntoDiPrelievo := ABS(IngombroSuperficialePinzaMAX * COS(deg_to_rad((ATAN(Larghezza/Lunghezza)*1/0.017+ Mission^.JPick))));
			(**************************************************************************************************************************************************)
			(* Ingombro ottimizzato della pinza sul punto di deposito *)
			(**************************************************************************************************************************************************)
			IngombroOttimizzatoX_InPuntoDiDeposito := ABS(IngombroSuperficialePinzaMAX * SIN(deg_to_rad((ATAN(Larghezza/Lunghezza)*1/0.017+ Mission^.JPlace))));
			IngombroOttimizzatoY_InPuntoDiDeposito := ABS(IngombroSuperficialePinzaMAX * COS(deg_to_rad((ATAN(Larghezza/Lunghezza)*1/0.017+ Mission^.JPlace))));
			*)			
			(**************************************************************************************************************************************************)
			(**************************************************************************************************************************************************)
			(* Valuto la direzione della X *)
			DirezioneXPositiva := TFDirezioneAssePositiva(Posizione_Attuale:=ModuleAX_X^.Ax^.Status.ActPosition,Posizione_Finale:=Mission^.XPlace);
			DirezioneXNegativa := NOT DirezioneXPositiva;
							
			(**************************************************************************************************************************************************)
			(* Ingombro MASSIMO della pinza durante il transito *)
			(**************************************************************************************************************************************************)
			//Calcolo ingombro attuale
			IF NOT TFAsseInFinestra(Posizione_Attuale:=ModuleAx_J^.Ax^.AxRef^.NcToPlc.ActPos,Posizione_Finale:=Mission^.JPlace,FinestraDiControllo:=5)  THEN //Se la pinza non è già nella finestra di destinazione 
				(* Calcolo l'ingombro massimo che assume durante il ciclo di lavoro nelle direzioni X e Y *)
				(*TFCalcoloIngombroOttimizzatoPinza(  Quota_RotazioneAttuale			:= ModuleAx_J^.Ax^.AxRef^.NcToPlc.ActPos,
													Quota_RotazioneDestinazione		:= Mission^.JPlace,
													IngombroSuperficialePinzaMAX	:= IngombroSuperficialePinzaMAX,
													Lunghezza						:= Larghezza,
													Larghezza						:= Lunghezza,
													IngombroOttimizzatoX_InTransito	=> IngombroOttimizzatoX_InTransito,
													IngombroOttimizzatoY_InTransito	=> IngombroOttimizzatoY_InTransito);*)
			ELSE;
				//IngombroOttimizzatoX_InTransito := ABS(IngombroSuperficialePinzaMAX * SIN(deg_to_rad((ATAN(Larghezza/Lunghezza)*1/0.017+ ModuleAx_J^.Ax^.AxRef^.NcToPlc.ActPos)))); //Ingombro Attuale direzione X
				//IngombroOttimizzatoY_InTransito := ABS(IngombroSuperficialePinzaMAX * COS(deg_to_rad((ATAN(Larghezza/Lunghezza)*1/0.017+ ModuleAx_J^.Ax^.AxRef^.NcToPlc.ActPos)))); //Ingombro Attuale direzione Y		
			END_IF
			(* Valutazione colonne in base al verso del pallettizzatore: verso stabilito guardando il pallettizzatore con la linea alle spalle *)
			CASE VERSO_PALLETTIZZATORE OF
				PALLETTIZZATORE_DX :
									TFCalcolaQuotaIngombroColonne(	QuotaY_ColonnaDX						:= WorkFootprint^[6].Y, //DX
																	QuotaY_ColonnaSX						:= WorkFootprint^[5].Y, //SX
																	QuotaAttualeAsse						:= ModuleAX_Y^.Ax^.AxRef^.NcToPlc.ActPos,
																	IngombroOttimizzatoY_InTransito         := IngombroOttimizzatoY_InTransito,
																	OffsetSicurezza_Y						:= OffsetSicurezza_Y,
																	QuotaDestinazioneAsse					:= Mission^.YPlace,
																	Pinza_InIngombroColonne_Attuale 		=> Pinza_InIngombroColonne_Attuale,
																	Pinza_InIngombroColonne_Destinazione 	=> Pinza_InIngombroColonne_Destinazione,
																	QuotaFuoriIngombro_Attuale_Y 			=> QuotaFuoriIngombro_Attuale_Y,
																	QuotaFuoriIngombro_Destinazione_Y 		=> QuotaFuoriIngombro_Destinazione_Y);
																	
				PALLETTIZZATORE_SX :
									TFCalcolaQuotaIngombroColonne(	QuotaY_ColonnaDX						:= WorkFootprint^[6].Y, //DX
																	QuotaY_ColonnaSX						:= WorkFootprint^[5].Y, //SX
																	QuotaAttualeAsse						:= ModuleAX_Y^.Ax^.AxRef^.NcToPlc.ActPos,
																	OffsetSicurezza_Y						:= OffsetSicurezza_Y,
																	IngombroOttimizzatoY_InTransito         := IngombroOttimizzatoY_InTransito,
																	QuotaDestinazioneAsse					:= Mission^.YPlace,
																	Pinza_InIngombroColonne_Attuale 		=> Pinza_InIngombroColonne_Attuale,
																	Pinza_InIngombroColonne_Destinazione 	=> Pinza_InIngombroColonne_Destinazione,
																	QuotaFuoriIngombro_Attuale_Y 			=> QuotaFuoriIngombro_Attuale_Y,
																	QuotaFuoriIngombro_Destinazione_Y 		=> QuotaFuoriIngombro_Destinazione_Y);
			END_CASE
			
			(* Setto la quota di fuori ingombro che la pinza dovrà assumere durante la traslazione per evitare la collisione con le colonne *)	
			QuotaFuoriIngombroColonne_Y := QuotaFuoriIngombro_Attuale_Y;
					
			(* Se sono in ingombro nella posizione attuale o nella posizione di destinazione, devo andare fuori-ingombro con la Y *)
			IF (Pinza_InIngombroColonne_Attuale OR Pinza_InIngombroColonne_Destinazione) THEN 
				IF (AsseXInFinestraDiRiposo AND AsseYInFinestraDiRiposo AND AsseJInFinestraDiRiposo) THEN //Se sono in finestra di riposo con tutti gli assi non devo andare fuori-ingombro con la Y
					FuoriIngombroYNecessarioTMP := FALSE;
				ELSE
					FuoriIngombroYNecessarioTMP := TRUE;
				END_IF
			ELSE
				FuoriIngombroYNecessarioTMP := FALSE;
			END_IF
		END_IF
			
	WAMANAGER_CICLO_DEPOSITO_FALDA_END:
		CalcolaIngombro := TRUE;	
(*
	WAMANAGER_CICLO_PACCO_INIT:
		CalcolaIngombro := TRUE;	
	
	WAMANAGER_CICLO_PRELIEVO_PACCO_RUN:
		DirezioneXPositiva := TFDirezioneAssePositiva(Posizione_Attuale:=ModuleAX_X^.Ax^.Status.ActPosition,Posizione_Finale:=Mission^.XPick);
		DirezioneXNegativa := NOT DirezioneXPositiva;
		(* Valuto se con l'asse X sono fuori dall'area delle colonne *)
		QuotaX_ConsensoRotazionePinza_Raggiunta := TFPinzaInFuoriIngombroColonne_DirezioneX(DirezioneXPositiva:=DirezioneXPositiva,
																							AsseInMoto:=ModuleAX_X^.Ax^.AxRef^.Status.Moving,
																							PosizioneAttuale:=ModuleAX_X^.Ax^.Status.ActPosition,
																							PosizioneColonna_X:=WorkFootprint^[5].X,  
																							IngombroColonna_X:=WorkFootprint^[5].XDim,
																							IngombroPinza_X:=IngombroX);																				
		
		IF CalcolaIngombro THEN
			CalcolaIngombro := FALSE;
			(* Definisco il tipo di area in cui si trova a lavorare il pallettizzatore *)
			AreaInLavoroPositiva := FALSE;
			AreaInLavoroNegativa := FALSE;
			AreaInLavoroPositivaNegativa := TRUE; 
			
			(**************************************************************************************************************************************************)
			(* Ingombro ottimizzato della pinza sul punto di prelievo *)
			(**************************************************************************************************************************************************)
			IngombroOttimizzatoX_InPuntoDiPrelievo := ABS(IngombroSuperficialePinzaMAX * SIN(deg_to_rad((ATAN(Larghezza/Lunghezza)*1/0.017+ Mission^.JPick))));
			IngombroOttimizzatoY_InPuntoDiPrelievo := ABS(IngombroSuperficialePinzaMAX * COS(deg_to_rad((ATAN(Larghezza/Lunghezza)*1/0.017+ Mission^.JPick))));
			(**************************************************************************************************************************************************)
			(* Ingombro ottimizzato della pinza sul punto di deposito *)
			(**************************************************************************************************************************************************)
			IngombroOttimizzatoX_InPuntoDiDeposito := ABS(IngombroSuperficialePinzaMAX * SIN(deg_to_rad((ATAN(Larghezza/Lunghezza)*1/0.017+ Mission^.JPlace))));
			IngombroOttimizzatoY_InPuntoDiDeposito := ABS(IngombroSuperficialePinzaMAX * COS(deg_to_rad((ATAN(Larghezza/Lunghezza)*1/0.017+ Mission^.JPlace))));
						
			(**************************************************************************************************************************************************)
			(**************************************************************************************************************************************************)
			(* Valuto la direzione della X *)
			DirezioneXPositiva := TFDirezioneAssePositiva(Posizione_Attuale:=ModuleAX_X^.Ax^.Status.ActPosition,Posizione_Finale:=Mission^.XPick);
			DirezioneXNegativa := NOT DirezioneXPositiva;
							
			(**************************************************************************************************************************************************)
			(* Ingombro MASSIMO della pinza durante il transito *)
			(**************************************************************************************************************************************************)
			//Calcolo ingombro attuale
			IF NOT TFAsseInFinestra(Posizione_Attuale:=ModuleAx_J^.Ax^.AxRef^.NcToPlc.ActPos,Posizione_Finale:=Mission^.JPick,FinestraDiControllo:=5)  THEN //Se la pinza non è già nella finestra di destinazione 
				(* Calcolo l'ingombro massimo che assume durante il ciclo di lavoro nelle direzioni X e Y *)
				TFCalcoloIngombroOttimizzatoPinza(  Quota_RotazioneAttuale			:= ModuleAx_J^.Ax^.AxRef^.NcToPlc.ActPos,
													Quota_RotazioneDestinazione		:= Mission^.JPick,
													IngombroSuperficialePinzaMAX	:= IngombroSuperficialePinzaMAX,
													Lunghezza						:= Larghezza,
													Larghezza						:= Lunghezza,
													IngombroOttimizzatoX_InTransito	=> IngombroOttimizzatoX_InTransito,
													IngombroOttimizzatoY_InTransito	=> IngombroOttimizzatoY_InTransito);
			ELSE
				IngombroOttimizzatoX_InTransito := ABS(IngombroSuperficialePinzaMAX * SIN(deg_to_rad((ATAN(Larghezza/Lunghezza)*1/0.017+ ModuleAx_J^.Ax^.AxRef^.NcToPlc.ActPos)))); //Ingombro Attuale direzione X
				IngombroOttimizzatoY_InTransito := ABS(IngombroSuperficialePinzaMAX * COS(deg_to_rad((ATAN(Larghezza/Lunghezza)*1/0.017+ ModuleAx_J^.Ax^.AxRef^.NcToPlc.ActPos)))); //Ingombro Attuale direzione Y		
			END_IF
			(* Valutazione colonne in base al verso del pallettizzatore: verso stabilito guardando il pallettizzatore con la linea alle spalle *)
			CASE VERSO_PALLETTIZZATORE OF
				PALLETTIZZATORE_DX :
									TFCalcolaQuotaIngombroColonne(	QuotaY_ColonnaDX						:= WorkFootprint^[6].Y, //DX
																	QuotaY_ColonnaSX						:= WorkFootprint^[5].Y, //SX
																	QuotaAttualeAsse						:= ModuleAX_Y^.Ax^.AxRef^.NcToPlc.ActPos,
																	IngombroOttimizzatoY_InTransito         := IngombroOttimizzatoY_InTransito,
																	OffsetSicurezza_Y						:= OffsetSicurezza_Y,
																	QuotaDestinazioneAsse					:= Mission^.YPick,
																	Pinza_InIngombroColonne_Attuale 		=> Pinza_InIngombroColonne_Attuale,
																	Pinza_InIngombroColonne_Destinazione 	=> Pinza_InIngombroColonne_Destinazione,
																	QuotaFuoriIngombro_Attuale_Y 			=> QuotaFuoriIngombro_Attuale_Y,
																	QuotaFuoriIngombro_Destinazione_Y 		=> QuotaFuoriIngombro_Destinazione_Y);
																	
				PALLETTIZZATORE_SX :
									TFCalcolaQuotaIngombroColonne(	QuotaY_ColonnaDX						:= WorkFootprint^[6].Y, //DX
																	QuotaY_ColonnaSX						:= WorkFootprint^[5].Y, //SX
																	QuotaAttualeAsse						:= ModuleAX_Y^.Ax^.AxRef^.NcToPlc.ActPos,
																	OffsetSicurezza_Y						:= OffsetSicurezza_Y,
																	IngombroOttimizzatoY_InTransito         := IngombroOttimizzatoY_InTransito,
																	QuotaDestinazioneAsse					:= Mission^.YPick,
																	Pinza_InIngombroColonne_Attuale 		=> Pinza_InIngombroColonne_Attuale,
																	Pinza_InIngombroColonne_Destinazione 	=> Pinza_InIngombroColonne_Destinazione,
																	QuotaFuoriIngombro_Attuale_Y 			=> QuotaFuoriIngombro_Attuale_Y,
																	QuotaFuoriIngombro_Destinazione_Y 		=> QuotaFuoriIngombro_Destinazione_Y);
			END_CASE
			
			(* Setto la quota di fuori ingombro che la pinza dovrà assumere durante la traslazione per evitare la collisione con le colonne *)	
			QuotaFuoriIngombroColonne_Y := QuotaFuoriIngombro_Attuale_Y;
					
			(* Se sono in ingombro nella posizione attuale o nella posizione di destinazione, devo andare fuori-ingombro con la Y *)
			IF (Pinza_InIngombroColonne_Attuale OR Pinza_InIngombroColonne_Destinazione) THEN 
				IF (AsseXInFinestraDiRiposo AND AsseYInFinestraDiRiposo AND AsseJInFinestraDiRiposo) THEN //Se sono in finestra di riposo con tutti gli assi non devo andare fuori-ingombro con la Y
					FuoriIngombroYNecessarioTMP := FALSE;
				ELSE
					FuoriIngombroYNecessarioTMP := TRUE;
				END_IF
			ELSE
				FuoriIngombroYNecessarioTMP := FALSE;
			END_IF
		END_IF
		
	WAMANAGER_CICLO_PRELIEVO_PACCO_END:
		CalcolaIngombro := TRUE;	
		
	WAMANAGER_CICLO_DEPOSITO_PACCO_RUN:
		DirezioneXPositiva := TFDirezioneAssePositiva(Posizione_Attuale:=ModuleAX_X^.Ax^.Status.ActPosition,Posizione_Finale:=Mission^.XPlace);
		DirezioneXNegativa := NOT DirezioneXPositiva;
		
		
		(* Larhezza Pick Point + Pacco *)
		(*IF WorkPickPointState^[1].XDim >= WorkPickPointDimension[1].XDim THEN
			LarghezzaPickPoint := WorkPickPointState^[1].XDim;
		else
			LarghezzaPickPoint := WorkPickPointDimension[1].Xdim;
		END_IF*)
				
		(* Valuto se con l'asse X sono fuori dall'area delle colonne *)
		QuotaX_ConsensoRotazionePinza_Raggiunta := TFPinzaInFuoriIngombroColonne_DirezioneX(DirezioneXPositiva:=DirezioneXPositiva,
																							AsseInMoto:=ModuleAX_X^.Ax^.AxRef^.Status.Moving,
																							PosizioneAttuale:=ModuleAX_X^.Ax^.Status.ActPosition,
																							PosizioneColonna_X:=WorkFootprint^[5].X,  
																							IngombroColonna_X:=WorkFootprint^[5].XDim,
																							IngombroPinza_X:=IngombroX);
		
		(*IF (WorkPickPoint^[Mission^.PPick].Xh >= WorkArea^[Mission^.PPlace].X AND Mission^.JPickVO = 1) OR 	//se il punto di prelievo IN ORRIZZONTALE ha quota maggiore della piazzola di deposito e
			(WorkPickPoint^[Mission^.PPick].Xv >= WorkArea^[Mission^.PPlace].X AND Mission^.JPickVO = 0) THEN
			 AreaInLavoroNegativa := TRUE;
		ELSIF (WorkPickPoint^[Mission^.PPick].Xh <= WorkArea^[Mission^.PPlace].X AND Mission^.JPickVO = 1) OR 	//se il punto di prelievo IN ORRIZZONTALE ha quota maggiore della piazzola di deposito e
			(WorkPickPoint^[Mission^.PPick].Xv <= WorkArea^[Mission^.PPlace].X AND Mission^.JPickVO = 0) THEN
			 AreaInLavoroPositiva := TRUE;
		END_IF*)																					
		CASE TIPO_RIBALTINO OF

			RIBALTINO_DOPO_SQUADRO:
									(* Valutazione Fuoringombro lungo X della pinza rispetto al ribaltino + Pacco*)
									IF (ModuleAX_X^.Ax^.Status.ActPosition + IngombroX/ 2 <= WorkPickPoint^[Mission^.PPick].Xv - LarghezzaPickPoint/2 + 30) OR 
										(ModuleAX_X^.Ax^.Status.ActPosition - IngombroX/ 2 >= WorkPickPoint^[Mission^.PPick].Xv + LarghezzaPickPoint/2 - 30) THEN
											QuotaFUPRINGOMBROdaRIBALTINO_X_RAGGIUNTA := TRUE;
									ELSE
										QuotaFUPRINGOMBROdaRIBALTINO_X_RAGGIUNTA := FALSE;
									END_IF
									
			RIBALTINO_DIRETTO:
							   (* Valutazione Fuoringombro lungo X della pinza rispetto al ribaltino + Pacco*)
								IF (ModuleAX_X^.Ax^.Status.ActPosition + IngombroX/ 2 <= WorkPickPoint^[Mission^.PPick].Xv + 30) OR 
									(ModuleAX_X^.Ax^.Status.ActPosition - IngombroX/ 2 >= WorkPickPoint^[Mission^.PPick].Xv - 30) THEN
										QuotaFUPRINGOMBROdaRIBALTINO_X_RAGGIUNTA := TRUE;
								ELSE
									QuotaFUPRINGOMBROdaRIBALTINO_X_RAGGIUNTA := FALSE;
								END_IF
								
								(* Valutazione Fuoringombro lungo Y della pinza rispetto al ribaltino + Pacco*)
								IF (ModuleAX_Y^.Ax^.Status.ActPosition + IngombroY/ 2 <= WorkPickPoint^[Mission^.PPick].Yv - LarghezzaPickPoint/2 + 30) OR 
									(ModuleAX_Y^.Ax^.Status.ActPosition - IngombroY/ 2 >= WorkPickPoint^[Mission^.PPick].Yv + LarghezzaPickPoint/2 - 30) OR
									(ModuleAX_Y^.Ax^.Status.ActPosition + IngombroY/ 2 <= WorkPickPoint^[Mission^.PPick].Yh - LarghezzaPickPoint/2 + 30) OR 
									(ModuleAX_Y^.Ax^.Status.ActPosition - IngombroY/ 2 >= WorkPickPoint^[Mission^.PPick].Yh + LarghezzaPickPoint/2 - 30) THEN
										QuotaFUPRINGOMBROdaRIBALTINO_Y_RAGGIUNTA := TRUE;
								ELSE
									QuotaFUPRINGOMBROdaRIBALTINO_Y_RAGGIUNTA := FALSE;
								END_IF
		END_CASE																	
																							
		IF CalcolaIngombro THEN
			CalcolaIngombro := FALSE;
			(* Definisco il tipo di area in cui si trova a lavorare il pallettizzatore *)
			AreaInLavoroPositiva := FALSE;
			AreaInLavoroNegativa := FALSE;
			AreaInLavoroPositivaNegativa := TRUE; 
			
			(**************************************************************************************************************************************************)
			(* Ingombro ottimizzato della pinza sul punto di prelievo *)
			(**************************************************************************************************************************************************)
			IngombroOttimizzatoX_InPuntoDiPrelievo := ABS(IngombroSuperficialePinzaMAX * SIN(deg_to_rad((ATAN(Larghezza/Lunghezza)*1/0.017+ Mission^.JPick))));
			IngombroOttimizzatoY_InPuntoDiPrelievo := ABS(IngombroSuperficialePinzaMAX * COS(deg_to_rad((ATAN(Larghezza/Lunghezza)*1/0.017+ Mission^.JPick))));
			(**************************************************************************************************************************************************)
			(* Ingombro ottimizzato della pinza sul punto di deposito *)
			(**************************************************************************************************************************************************)
			IngombroOttimizzatoX_InPuntoDiDeposito := ABS(IngombroSuperficialePinzaMAX * SIN(deg_to_rad((ATAN(Larghezza/Lunghezza)*1/0.017+ Mission^.JPlace))));
			IngombroOttimizzatoY_InPuntoDiDeposito := ABS(IngombroSuperficialePinzaMAX * COS(deg_to_rad((ATAN(Larghezza/Lunghezza)*1/0.017+ Mission^.JPlace))));
						
			(**************************************************************************************************************************************************)
			(**************************************************************************************************************************************************)
			(* Valuto la direzione della X *)
			DirezioneXPositiva := TFDirezioneAssePositiva(Posizione_Attuale:=ModuleAX_X^.Ax^.Status.ActPosition,Posizione_Finale:=Mission^.XPlace);
			DirezioneXNegativa := NOT DirezioneXPositiva;
							
			(**************************************************************************************************************************************************)
			(* Ingombro MASSIMO della pinza durante il transito *)
			(**************************************************************************************************************************************************)
			//Calcolo ingombro attuale
			IF NOT TFAsseInFinestra(Posizione_Attuale:=ModuleAx_J^.Ax^.AxRef^.NcToPlc.ActPos,Posizione_Finale:=Mission^.JPlace,FinestraDiControllo:=5)  THEN //Se la pinza non è già nella finestra di destinazione 
				(* Calcolo l'ingombro massimo che assume durante il ciclo di lavoro nelle direzioni X e Y *)
				TFCalcoloIngombroOttimizzatoPinza(  Quota_RotazioneAttuale			:= ModuleAx_J^.Ax^.AxRef^.NcToPlc.ActPos,
													Quota_RotazioneDestinazione		:= Mission^.JPlace,
													IngombroSuperficialePinzaMAX	:= IngombroSuperficialePinzaMAX,
													Lunghezza						:= Larghezza,
													Larghezza						:= Lunghezza,
													IngombroOttimizzatoX_InTransito	=> IngombroOttimizzatoX_InTransito,
													IngombroOttimizzatoY_InTransito	=> IngombroOttimizzatoY_InTransito);
			ELSE
				IngombroOttimizzatoX_InTransito := ABS(IngombroSuperficialePinzaMAX * SIN(deg_to_rad((ATAN(Larghezza/Lunghezza)*1/0.017+ ModuleAx_J^.Ax^.AxRef^.NcToPlc.ActPos)))); //Ingombro Attuale direzione X
				IngombroOttimizzatoY_InTransito := ABS(IngombroSuperficialePinzaMAX * COS(deg_to_rad((ATAN(Larghezza/Lunghezza)*1/0.017+ ModuleAx_J^.Ax^.AxRef^.NcToPlc.ActPos)))); //Ingombro Attuale direzione Y		
			END_IF
			(* Valutazione colonne in base al verso del pallettizzatore: verso stabilito guardando il pallettizzatore con la linea alle spalle *)
			CASE VERSO_PALLETTIZZATORE OF
				PALLETTIZZATORE_DX :
									TFCalcolaQuotaIngombroColonne(	QuotaY_ColonnaDX						:= WorkFootprint^[6].Y, //DX
																	QuotaY_ColonnaSX						:= WorkFootprint^[5].Y, //SX
																	QuotaAttualeAsse						:= ModuleAX_Y^.Ax^.AxRef^.NcToPlc.ActPos,
																	IngombroOttimizzatoY_InTransito         := IngombroOttimizzatoY_InTransito,
																	OffsetSicurezza_Y						:= OffsetSicurezza_Y,
																	QuotaDestinazioneAsse					:= Mission^.YPlace,
																	Pinza_InIngombroColonne_Attuale 		=> Pinza_InIngombroColonne_Attuale,
																	Pinza_InIngombroColonne_Destinazione 	=> Pinza_InIngombroColonne_Destinazione,
																	QuotaFuoriIngombro_Attuale_Y 			=> QuotaFuoriIngombro_Attuale_Y,
																	QuotaFuoriIngombro_Destinazione_Y 		=> QuotaFuoriIngombro_Destinazione_Y);
																	
				PALLETTIZZATORE_SX :
									TFCalcolaQuotaIngombroColonne(	QuotaY_ColonnaDX						:= WorkFootprint^[6].Y, //DX
																	QuotaY_ColonnaSX						:= WorkFootprint^[5].Y, //SX
																	QuotaAttualeAsse						:= ModuleAX_Y^.Ax^.AxRef^.NcToPlc.ActPos,
																	OffsetSicurezza_Y						:= OffsetSicurezza_Y,
																	IngombroOttimizzatoY_InTransito         := IngombroOttimizzatoY_InTransito,
																	QuotaDestinazioneAsse					:= Mission^.YPlace,
																	Pinza_InIngombroColonne_Attuale 		=> Pinza_InIngombroColonne_Attuale,
																	Pinza_InIngombroColonne_Destinazione 	=> Pinza_InIngombroColonne_Destinazione,
																	QuotaFuoriIngombro_Attuale_Y 			=> QuotaFuoriIngombro_Attuale_Y,
																	QuotaFuoriIngombro_Destinazione_Y 		=> QuotaFuoriIngombro_Destinazione_Y);
			END_CASE
			
			(* Setto la quota di fuori ingombro che la pinza dovrà assumere durante la traslazione per evitare la collisione con le colonne *)	
			QuotaFuoriIngombroColonne_Y := QuotaFuoriIngombro_Attuale_Y;
					
			(* Se sono in ingombro nella posizione attuale o nella posizione di destinazione, devo andare fuori-ingombro con la Y *)
			IF (Pinza_InIngombroColonne_Attuale OR Pinza_InIngombroColonne_Destinazione) THEN 
				IF (AsseXInFinestraDiRiposo AND AsseYInFinestraDiRiposo AND AsseJInFinestraDiRiposo) THEN //Se sono in finestra di riposo con tutti gli assi non devo andare fuori-ingombro con la Y
					FuoriIngombroYNecessarioTMP := FALSE;
				ELSE
					FuoriIngombroYNecessarioTMP := TRUE;
				END_IF
			ELSE
				FuoriIngombroYNecessarioTMP := FALSE;
			END_IF
		END_IF
		
	WAMANAGER_CICLO_DEPOSITO_PACCO_END:
		CalcolaIngombro := TRUE;	*)
	
END_CASE

END_FUNCTION_BLOCK

(* stored: Version 1.1.0.1, ProductVersion 3.1.4024.11
   POU TFCalcoliFuoriIngombriColonne: Id {5698b144-3aba-4d90-82ff-8ae0b80dc9b7}, SpecialFunc None *)
